		IF fbSQLDatabaseEvt.CreateSP('[dbo].[GetResourcesByNameMilling]', ADR(SQLSPParameterSize1), SIZEOF(SQLSPParameterSize1), pSQLStoredProcedureEvt[29]) THEN	
			IF fbSQLDatabaseEvt.bError THEN
    	
				iState							:=1340;
			ELSE
				
				iState							:= 350;
			END_IF
		END_IF
		
	350:
		SQLSPParameterSize3[0].sParameterName := '@return';
		SQLSPParameterSize3[0].eParameterType := E_SPParameterType.ReturnValue;
		SQLSPParameterSize3[0].eParameterDataType := E_ColumnType.Integer;
		SQLSPParameterSize3[0].nParameterSize := SIZEOF(DINT);
	
		SQLSPParameterSize3[1].sParameterName := '@StatusFilter';
		SQLSPParameterSize3[1].eParameterType := E_SPParameterType.Input;
		SQLSPParameterSize3[1].eParameterDataType := E_ColumnType.NVarChar;
		SQLSPParameterSize3[1].nParameterSize := SIZEOF(STRING(50));
		                  
		SQLSPParameterSize3[2].sParameterName := '@OrderListJson';
		SQLSPParameterSize3[2].eParameterType := E_SPParameterType.Output;
		SQLSPParameterSize3[2].eParameterDataType := E_ColumnType.NVarChar;
		SQLSPParameterSize3[2].nParameterSize := SIZEOF(STRING(DB.MAX_STRING_SIZE));
		
		IF fbSQLDatabaseEvt.CreateSP('[dbo].[MES_GetOrderInfoList]', ADR(SQLSPParameterSize3), SIZEOF(SQLSPParameterSize3), pSQLStoredProcedureEvt[31]) THEN	
			IF fbSQLDatabaseEvt.bError THEN
    	
				iState							:=1350;
			ELSE
				
				iState							:= 360;
			END_IF
		END_IF	
		
	360:
		SQLSPParameterSize3[0].sParameterName := '@return';
		SQLSPParameterSize3[0].eParameterType := E_SPParameterType.ReturnValue;
		SQLSPParameterSize3[0].eParameterDataType := E_ColumnType.Integer;
		SQLSPParameterSize3[0].nParameterSize := SIZEOF(DINT);
	
		SQLSPParameterSize3[1].sParameterName := '@OrderReference';
		SQLSPParameterSize3[1].eParameterType := E_SPParameterType.Input;
		SQLSPParameterSize3[1].eParameterDataType := E_ColumnType.NVarChar;
		SQLSPParameterSize3[1].nParameterSize := SIZEOF(STRING(50));
		                  
		SQLSPParameterSize3[2].sParameterName := '@OrderItemsJson';
		SQLSPParameterSize3[2].eParameterType := E_SPParameterType.Output;
		SQLSPParameterSize3[2].eParameterDataType := E_ColumnType.NVarChar;
		SQLSPParameterSize3[2].nParameterSize := SIZEOF(STRING(DB.MAX_STRING_SIZE));
		
		IF fbSQLDatabaseEvt.CreateSP('[dbo].[MES_GetOrderItems]', ADR(SQLSPParameterSize3), SIZEOF(SQLSPParameterSize3), pSQLStoredProcedureEvt[32]) THEN	
			IF fbSQLDatabaseEvt.bError THEN
    	
				iState							:=1360;
			ELSE
				
				iState							:= 370;
			END_IF
		END_IF	
		
	370:
		SQLSPParameterSize2[0].sParameterName := '@return';
		SQLSPParameterSize2[0].eParameterType := E_SPParameterType.ReturnValue;
		SQLSPParameterSize2[0].eParameterDataType := E_ColumnType.Integer;
		SQLSPParameterSize2[0].nParameterSize := SIZEOF(DINT);
	                      
		SQLSPParameterSize2[1].sParameterName := '@BatchId';
		SQLSPParameterSize2[1].eParameterType := E_SPParameterType.Input;
		SQLSPParameterSize2[1].eParameterDataType := E_ColumnType.NVarChar;
		SQLSPParameterSize2[1].nParameterSize := SIZEOF(STRING(50));
		
		IF fbSQLDatabaseEvt.CreateSP('[dbo].[GetOrderItems]', ADR(SQLSPParameterSize2), SIZEOF(SQLSPParameterSize2), pSQLStoredProcedureEvt[33]) THEN	
			IF fbSQLDatabaseEvt.bError THEN
    	
				iState							:=1370;
			ELSE
				
				iState							:= 380;
			END_IF
		END_IF	
		
	380:
		SQLSPParameterSize3[0].sParameterName := '@return';
		SQLSPParameterSize3[0].eParameterType := E_SPParameterType.ReturnValue;
		SQLSPParameterSize3[0].eParameterDataType := E_ColumnType.Integer;
		SQLSPParameterSize3[0].nParameterSize := SIZEOF(DINT);
	                      
		SQLSPParameterSize3[1].sParameterName := '@InputJson';
		SQLSPParameterSize3[1].eParameterType := E_SPParameterType.Input;
		SQLSPParameterSize3[1].eParameterDataType := E_ColumnType.NVarChar;
		SQLSPParameterSize3[1].nParameterSize := SIZEOF(STRING(DB.MAX_STRING_SIZE));
		
		SQLSPParameterSize3[2].sParameterName := '@OutputJson';
		SQLSPParameterSize3[2].eParameterType := E_SPParameterType.Output;
		SQLSPParameterSize3[2].eParameterDataType := E_ColumnType.NVarChar;
		SQLSPParameterSize3[2].nParameterSize := SIZEOF(STRING(DB.MAX_STRING_SIZE));
	
		IF fbSQLDatabaseEvt.CreateSP('[dbo].[GetBatchList]', ADR(SQLSPParameterSize3), SIZEOF(SQLSPParameterSize3), pSQLStoredProcedureEvt[34]) THEN	
			IF fbSQLDatabaseEvt.bError THEN
    	
				iState							:=1380;
			ELSE
				
				iState							:= 390;
			END_IF
		END_IF
		
	390:
		SQLSPParameterSize3[0].sParameterName := '@return';
		SQLSPParameterSize3[0].eParameterType := E_SPParameterType.ReturnValue;
		SQLSPParameterSize3[0].eParameterDataType := E_ColumnType.Integer;
		SQLSPParameterSize3[0].nParameterSize := SIZEOF(DINT);
	                      
		SQLSPParameterSize3[1].sParameterName := '@InputJson';
		SQLSPParameterSize3[1].eParameterType := E_SPParameterType.Input;
		SQLSPParameterSize3[1].eParameterDataType := E_ColumnType.NVarChar;
		SQLSPParameterSize3[1].nParameterSize := SIZEOF(STRING(DB.MAX_STRING_SIZE));
		
		SQLSPParameterSize3[2].sParameterName := '@OutputJson';
		SQLSPParameterSize3[2].eParameterType := E_SPParameterType.Output;
		SQLSPParameterSize3[2].eParameterDataType := E_ColumnType.NVarChar;
		SQLSPParameterSize3[2].nParameterSize := SIZEOF(STRING(DB.MAX_STRING_SIZE));
	
		IF fbSQLDatabaseEvt.CreateSP('[dbo].[GetBatchList]', ADR(SQLSPParameterSize3), SIZEOF(SQLSPParameterSize3), pSQLStoredProcedureEvt[35]) THEN	
			IF fbSQLDatabaseEvt.bError THEN
    	
				iState							:=1390;
			ELSE
				
				iState							:= 400;
			END_IF
		END_IF
		
	400:
		SQLSPParameterSize1[0].sParameterName := '@return';
		SQLSPParameterSize1[0].eParameterType := E_SPParameterType.ReturnValue;
		SQLSPParameterSize1[0].eParameterDataType := E_ColumnType.Integer;
		SQLSPParameterSize1[0].nParameterSize := SIZEOF(DINT);
		
		IF fbSQLDatabaseEvt.CreateSP('[dbo].[CMD_AbortProduction]', ADR(SQLSPParameterSize1), SIZEOF(SQLSPParameterSize1), pSQLStoredProcedureEvt[36]) THEN	
			IF fbSQLDatabaseEvt.bError THEN
    	
				iState							:=1400;
			ELSE
				
				iState							:= 410;
			END_IF
		END_IF
		
	410:
		SQLSPParameterSize3[0].sParameterName := '@return';
		SQLSPParameterSize3[0].eParameterType := E_SPParameterType.ReturnValue;
		SQLSPParameterSize3[0].eParameterDataType := E_ColumnType.Integer;
		SQLSPParameterSize3[0].nParameterSize := SIZEOF(DINT);
		                  
		SQLSPParameterSize3[1].sParameterName := '@currentPage';
		SQLSPParameterSize3[1].eParameterType := E_SPParameterType.Input;
		SQLSPParameterSize3[1].eParameterDataType := E_ColumnType.Integer;
		SQLSPParameterSize3[1].nParameterSize := SIZEOF(DINT);
		                  
		SQLSPParameterSize3[2].sParameterName := '@recordToFetch';
		SQLSPParameterSize3[2].eParameterType := E_SPParameterType.Input;
		SQLSPParameterSize3[2].eParameterDataType := E_ColumnType.Integer;
		SQLSPParameterSize3[2].nParameterSize := SIZEOF(DINT);
		
		IF fbSQLDatabaseEvt.CreateSP('[dbo].[GetBatchHistory]', ADR(SQLSPParameterSize3), SIZEOF(SQLSPParameterSize3), pSQLStoredProcedureEvt[37]) THEN	
			IF fbSQLDatabaseEvt.bError THEN
    	
				iState							:=1410;
			ELSE
				
				iState							:= 420;
			END_IF
		END_IF

	420:
		SQLSPParameterSize2[0].sParameterName := '@return';
		SQLSPParameterSize2[0].eParameterType := E_SPParameterType.ReturnValue;
		SQLSPParameterSize2[0].eParameterDataType := E_ColumnType.Integer;
		SQLSPParameterSize2[0].nParameterSize := SIZEOF(DINT);

		SQLSPParameterSize2[1].sParameterName := '@BatchId';
		SQLSPParameterSize2[1].eParameterType := E_SPParameterType.Input;
		SQLSPParameterSize2[1].eParameterDataType := E_ColumnType.NVarChar;
		SQLSPParameterSize2[1].nParameterSize := SIZEOF(STRING(50));
		
		IF fbSQLDatabaseEvt.CreateSP('[dbo].[GetBatchHistoryDetail]', ADR(SQLSPParameterSize2), SIZEOF(SQLSPParameterSize2), pSQLStoredProcedureEvt[38]) THEN	
			IF fbSQLDatabaseEvt.bError THEN
    	
				iState							:=1420;
			ELSE
				
				iState							:= 430;
			END_IF
		END_IF
		
	430:
		SQLSPParameterSize2[0].sParameterName := '@return';
		SQLSPParameterSize2[0].eParameterType := E_SPParameterType.ReturnValue;
		SQLSPParameterSize2[0].eParameterDataType := E_ColumnType.Integer;
		SQLSPParameterSize2[0].nParameterSize := SIZEOF(DINT);

		SQLSPParameterSize2[1].sParameterName := '@Id';
		SQLSPParameterSize2[1].eParameterType := E_SPParameterType.Input;
		SQLSPParameterSize2[1].eParameterDataType := E_ColumnType.NVarChar;
		SQLSPParameterSize2[1].nParameterSize := SIZEOF(STRING(50));
		
		IF fbSQLDatabaseEvt.CreateSP('[dbo].[CMD_ForceCompletedBatch]', ADR(SQLSPParameterSize2), SIZEOF(SQLSPParameterSize2), pSQLStoredProcedureEvt[39]) THEN	
			IF fbSQLDatabaseEvt.bError THEN
    	
				iState							:=1430;
			ELSE
				
				iState							:= 440;
			END_IF
		END_IF
		
	440:
		SQLSPParameterSize2[0].sParameterName := '@return';
		SQLSPParameterSize2[0].eParameterType := E_SPParameterType.ReturnValue;
		SQLSPParameterSize2[0].eParameterDataType := E_ColumnType.Integer;
		SQLSPParameterSize2[0].nParameterSize := SIZEOF(DINT);

		SQLSPParameterSize2[1].sParameterName := '@Id';
		SQLSPParameterSize2[1].eParameterType := E_SPParameterType.Input;
		SQLSPParameterSize2[1].eParameterDataType := E_ColumnType.NVarChar;
		SQLSPParameterSize2[1].nParameterSize := SIZEOF(STRING(50));
		
		IF fbSQLDatabaseEvt.CreateSP('[dbo].[CMD_HoldBatch]', ADR(SQLSPParameterSize2), SIZEOF(SQLSPParameterSize2), pSQLStoredProcedureEvt[40]) THEN	
			IF fbSQLDatabaseEvt.bError THEN
    	
				iState							:=1440;
			ELSE
				
				iState							:= 450;
			END_IF
		END_IF
		
	450:
		SQLSPParameterSize3[0].sParameterName := '@return';
		SQLSPParameterSize3[0].eParameterType := E_SPParameterType.ReturnValue;
		SQLSPParameterSize3[0].eParameterDataType := E_ColumnType.Integer;
		SQLSPParameterSize3[0].nParameterSize := SIZEOF(DINT);
                          
		SQLSPParameterSize3[1].sParameterName := '@Id';
		SQLSPParameterSize3[1].eParameterType := E_SPParameterType.Input;
		SQLSPParameterSize3[1].eParameterDataType := E_ColumnType.NVarChar;
		SQLSPParameterSize3[1].nParameterSize := SIZEOF(STRING(50));
		
		SQLSPParameterSize3[2].sParameterName := '@Mode';
		SQLSPParameterSize3[2].eParameterType := E_SPParameterType.Input;
		SQLSPParameterSize3[2].eParameterDataType := E_ColumnType.NVarChar;
		SQLSPParameterSize3[2].nParameterSize := SIZEOF(STRING(50));
		
		IF fbSQLDatabaseEvt.CreateSP('[dbo].[CMD_RecoverBatch]', ADR(SQLSPParameterSize3), SIZEOF(SQLSPParameterSize3), pSQLStoredProcedureEvt[41]) THEN	
			IF fbSQLDatabaseEvt.bError THEN
    	
				iState							:=1450;
			ELSE
				
				iState							:= 460;
			END_IF
		END_IF
		
	460:
		SQLSPParameterSize4[0].sParameterName := '@return';
		SQLSPParameterSize4[0].eParameterType := E_SPParameterType.ReturnValue;
		SQLSPParameterSize4[0].eParameterDataType := E_ColumnType.Integer;
		SQLSPParameterSize4[0].nParameterSize := SIZEOF(DINT);
                          
		SQLSPParameterSize4[1].sParameterName := '@Id';
		SQLSPParameterSize4[1].eParameterType := E_SPParameterType.Input;
		SQLSPParameterSize4[1].eParameterDataType := E_ColumnType.NVarChar;
		SQLSPParameterSize4[1].nParameterSize := SIZEOF(STRING(50));
		                  
		SQLSPParameterSize4[2].sParameterName := '@Mode';
		SQLSPParameterSize4[2].eParameterType := E_SPParameterType.Input;
		SQLSPParameterSize4[2].eParameterDataType := E_ColumnType.NVarChar;
		SQLSPParameterSize4[2].nParameterSize := SIZEOF(STRING(50));
		                  
		SQLSPParameterSize4[3].sParameterName := '@RestartMode';
		SQLSPParameterSize4[3].eParameterType := E_SPParameterType.Input;
		SQLSPParameterSize4[3].eParameterDataType := E_ColumnType.NVarChar;
		SQLSPParameterSize4[3].nParameterSize := SIZEOF(STRING(50));
		
		IF fbSQLDatabaseEvt.CreateSP('[dbo].[CMD_RestartBatch]', ADR(SQLSPParameterSize4), SIZEOF(SQLSPParameterSize4), pSQLStoredProcedureEvt[42]) THEN	
			IF fbSQLDatabaseEvt.bError THEN
    	
				iState							:=1460;
			ELSE
				
				iState							:= 470;
			END_IF
		END_IF
		
	470:
		SQLSPParameterSize3[0].sParameterName := '@return';
		SQLSPParameterSize3[0].eParameterType := E_SPParameterType.ReturnValue;
		SQLSPParameterSize3[0].eParameterDataType := E_ColumnType.Integer;
		SQLSPParameterSize3[0].nParameterSize := SIZEOF(DINT);
                          
		SQLSPParameterSize3[1].sParameterName := '@Id';
		SQLSPParameterSize3[1].eParameterType := E_SPParameterType.Input;
		SQLSPParameterSize3[1].eParameterDataType := E_ColumnType.NVarChar;
		SQLSPParameterSize3[1].nParameterSize := SIZEOF(STRING(50));
		
		SQLSPParameterSize3[2].sParameterName := '@Mode';
		SQLSPParameterSize3[2].eParameterType := E_SPParameterType.Input;
		SQLSPParameterSize3[2].eParameterDataType := E_ColumnType.NVarChar;
		SQLSPParameterSize3[2].nParameterSize := SIZEOF(STRING(50));
		
		IF fbSQLDatabaseEvt.CreateSP('[dbo].[CMD_ResumeBatch]', ADR(SQLSPParameterSize3), SIZEOF(SQLSPParameterSize3), pSQLStoredProcedureEvt[43]) THEN	
			IF fbSQLDatabaseEvt.bError THEN
    	
				iState							:=1470;
			ELSE
				
				iState							:= 480;
			END_IF
		END_IF
		
	480:
		SQLSPParameterSize3[0].sParameterName := '@return';
		SQLSPParameterSize3[0].eParameterType := E_SPParameterType.ReturnValue;
		SQLSPParameterSize3[0].eParameterDataType := E_ColumnType.Integer;
		SQLSPParameterSize3[0].nParameterSize := SIZEOF(DINT);
                          
		SQLSPParameterSize3[1].sParameterName := '@Id';
		SQLSPParameterSize3[1].eParameterType := E_SPParameterType.Input;
		SQLSPParameterSize3[1].eParameterDataType := E_ColumnType.NVarChar;
		SQLSPParameterSize3[1].nParameterSize := SIZEOF(STRING(50));
		
		SQLSPParameterSize3[2].sParameterName := '@Mode';
		SQLSPParameterSize3[2].eParameterType := E_SPParameterType.Input;
		SQLSPParameterSize3[2].eParameterDataType := E_ColumnType.NVarChar;
		SQLSPParameterSize3[2].nParameterSize := SIZEOF(STRING(50));
		
		IF fbSQLDatabaseEvt.CreateSP('[dbo].[CMD_SuspendBatch]', ADR(SQLSPParameterSize3), SIZEOF(SQLSPParameterSize3), pSQLStoredProcedureEvt[44]) THEN	
			IF fbSQLDatabaseEvt.bError THEN
    	
				iState							:=1480;
			ELSE
				
				iState							:= 490;
			END_IF
		END_IF
		
	490:
		SQLSPParameterSize2[0].sParameterName := '@return';
		SQLSPParameterSize2[0].eParameterType := E_SPParameterType.ReturnValue;
		SQLSPParameterSize2[0].eParameterDataType := E_ColumnType.Integer;
		SQLSPParameterSize2[0].nParameterSize := SIZEOF(DINT);

		SQLSPParameterSize2[1].sParameterName := '@Id';
		SQLSPParameterSize2[1].eParameterType := E_SPParameterType.Input;
		SQLSPParameterSize2[1].eParameterDataType := E_ColumnType.NVarChar;
		SQLSPParameterSize2[1].nParameterSize := SIZEOF(STRING(50));
		
		IF fbSQLDatabaseEvt.CreateSP('[dbo].[CMD_UnholdBatch]', ADR(SQLSPParameterSize2), SIZEOF(SQLSPParameterSize2), pSQLStoredProcedureEvt[45]) THEN	
			IF fbSQLDatabaseEvt.bError THEN
    	
				iState							:=1490;
			ELSE
				
				iState							:= 500;
			END_IF
		END_IF

	500:
		SQLSPParameterSize3[0].sParameterName := '@return';
		SQLSPParameterSize3[0].eParameterType := E_SPParameterType.ReturnValue;
		SQLSPParameterSize3[0].eParameterDataType := E_ColumnType.Integer;
		SQLSPParameterSize3[0].nParameterSize := SIZEOF(DINT);

		SQLSPParameterSize3[1].sParameterName := '@Name';
		SQLSPParameterSize3[1].eParameterType := E_SPParameterType.Input;
		SQLSPParameterSize3[1].eParameterDataType := E_ColumnType.NVarChar;
		SQLSPParameterSize3[1].nParameterSize := SIZEOF(STRING(50));
		
		SQLSPParameterSize3[2].sParameterName := '@JsonValue';
		SQLSPParameterSize3[2].eParameterType := E_SPParameterType.Input;
		SQLSPParameterSize3[2].eParameterDataType := E_ColumnType.NVarChar;
		SQLSPParameterSize3[2].nParameterSize := SIZEOF(STRING(DB.MAX_STRING_SIZE));
		
		IF fbSQLDatabaseEvt.CreateSP('[dbo].[UpdateSettingRepositoryByName]', ADR(SQLSPParameterSize3), SIZEOF(SQLSPParameterSize3), pSQLStoredProcedureEvt[46]) THEN	
			IF fbSQLDatabaseEvt.bError THEN
    	
				iState							:=1500;
			ELSE
				
				iState							:= 510;
			END_IF
		END_IF		
	
	510:
		SQLSPParameterSize1[0].sParameterName := '@return';
		SQLSPParameterSize1[0].eParameterType := E_SPParameterType.ReturnValue;
		SQLSPParameterSize1[0].eParameterDataType := E_ColumnType.Integer;
		SQLSPParameterSize1[0].nParameterSize := SIZEOF(DINT);
		
		IF fbSQLDatabaseEvt.CreateSP('[dbo].[GetSettingRepositoryList]', ADR(SQLSPParameterSize1), SIZEOF(SQLSPParameterSize1), pSQLStoredProcedureEvt[47]) THEN	
			IF fbSQLDatabaseEvt.bError THEN
    	
				iState							:=1510;
			ELSE
				
				iState							:= 520;
			END_IF
		END_IF	
		
	520:
		SQLSPParameterSize2[0].sParameterName := '@return';
		SQLSPParameterSize2[0].eParameterType := E_SPParameterType.ReturnValue;
		SQLSPParameterSize2[0].eParameterDataType := E_ColumnType.Integer;
		SQLSPParameterSize2[0].nParameterSize := SIZEOF(DINT);

		SQLSPParameterSize2[1].sParameterName := '@BatchId';
		SQLSPParameterSize2[1].eParameterType := E_SPParameterType.Input;
		SQLSPParameterSize2[1].eParameterDataType := E_ColumnType.NVarChar;
		SQLSPParameterSize2[1].nParameterSize := SIZEOF(STRING(50));
		
		IF fbSQLDatabaseEvt.CreateSP('[dbo].[GetBatchDetailById]', ADR(SQLSPParameterSize2), SIZEOF(SQLSPParameterSize2), pSQLStoredProcedureEvt[48]) THEN	
			IF fbSQLDatabaseEvt.bError THEN
    	
				iState							:=1520;
			ELSE
				
				iState							:=530;
			END_IF
		END_IF
		
	530:
		SQLSPParameterSize3[0].sParameterName := '@return';
		SQLSPParameterSize3[0].eParameterType := E_SPParameterType.ReturnValue;
		SQLSPParameterSize3[0].eParameterDataType := E_ColumnType.Integer;
		SQLSPParameterSize3[0].nParameterSize := SIZEOF(DINT);

		SQLSPParameterSize3[1].sParameterName := '@BatchId';
		SQLSPParameterSize3[1].eParameterType := E_SPParameterType.Input;
		SQLSPParameterSize3[1].eParameterDataType := E_ColumnType.NVarChar;
		SQLSPParameterSize3[1].nParameterSize := SIZEOF(STRING(50));
		
		SQLSPParameterSize3[2].sParameterName := '@DestinationPosition';
		SQLSPParameterSize3[2].eParameterType := E_SPParameterType.Input;
		SQLSPParameterSize3[2].eParameterDataType := E_ColumnType.Integer;
		SQLSPParameterSize3[2].nParameterSize := SIZEOF(DINT);
		
		IF fbSQLDatabaseEvt.CreateSP('[dbo].[ChangeBatchPositionInProductionQueue]', ADR(SQLSPParameterSize3), SIZEOF(SQLSPParameterSize3), pSQLStoredProcedureEvt[49]) THEN	
			IF fbSQLDatabaseEvt.bError THEN
    	
				iState							:=1530;
			ELSE
				
				iState							:= 540;
			END_IF
		END_IF
		
	540:
		SQLSPParameterSize2[0].sParameterName := '@Drum';
		SQLSPParameterSize2[0].eParameterType := E_SPParameterType.Input;
		SQLSPParameterSize2[0].eParameterDataType := E_ColumnType.NVarChar;
		SQLSPParameterSize2[0].nParameterSize := SIZEOF(STRING(30));	
	                      
		SQLSPParameterSize2[1].sParameterName := '@JsonResult';
		SQLSPParameterSize2[1].eParameterType := E_SPParameterType.Output;
		SQLSPParameterSize2[1].eParameterDataType := E_ColumnType.NVarChar;
		SQLSPParameterSize2[1].nParameterSize := SIZEOF(STRING(DB.MAX_STRING_SIZE));
	
		IF fbSQLDatabaseEvt.CreateSP('[dbo].[GetCuttersOnDrum]', ADR(SQLSPParameterSize2), SIZEOF(SQLSPParameterSize2), pSQLStoredProcedureEvt[50]) THEN	
			IF fbSQLDatabaseEvt.bError THEN
    	
				iState							:=1540;
			ELSE
				
				iState							:= 550;
			END_IF
		END_IF
		
	550:
		SQLSPParameterSize1[0].sParameterName := '@JsonResult';
		SQLSPParameterSize1[0].eParameterType := E_SPParameterType.Output;
		SQLSPParameterSize1[0].eParameterDataType := E_ColumnType.NVarChar;
		SQLSPParameterSize1[0].nParameterSize := SIZEOF(STRING(DB.MAX_STRING_SIZE));
	
		IF fbSQLDatabaseEvt.CreateSP('[dbo].[GetCuttersComboboxFormatted]', ADR(SQLSPParameterSize1), SIZEOF(SQLSPParameterSize1), pSQLStoredProcedureEvt[51]) THEN	
			IF fbSQLDatabaseEvt.bError THEN
    	
				iState							:=1550;
			ELSE
				
				iState							:= 560;
			END_IF
		END_IF
		
	560:
		SQLSPParameterSize2[0].sParameterName := '@Drum';
		SQLSPParameterSize2[0].eParameterType := E_SPParameterType.Input;
		SQLSPParameterSize2[0].eParameterDataType := E_ColumnType.NVarChar;
		SQLSPParameterSize2[0].nParameterSize := SIZEOF(STRING(30));	
	                      
		SQLSPParameterSize2[1].sParameterName := '@JsonValue';
		SQLSPParameterSize2[1].eParameterType := E_SPParameterType.Input;
		SQLSPParameterSize2[1].eParameterDataType := E_ColumnType.NVarChar;
		SQLSPParameterSize2[1].nParameterSize := SIZEOF(STRING(DB.MAX_STRING_SIZE));
	
		IF fbSQLDatabaseEvt.CreateSP('[dbo].[UpdateCuttersOnDrum]', ADR(SQLSPParameterSize2), SIZEOF(SQLSPParameterSize2), pSQLStoredProcedureEvt[52]) THEN	
			IF fbSQLDatabaseEvt.bError THEN
    	
				iState							:=1560;
			ELSE
				
				iState							:= 570;
			END_IF
		END_IF
		
	570:
		SQLSPParameterSize3[0].sParameterName := '@Id';
		SQLSPParameterSize3[0].eParameterType := E_SPParameterType.Input;
		SQLSPParameterSize3[0].eParameterDataType := E_ColumnType.Integer;
		SQLSPParameterSize3[0].nParameterSize := SIZEOF(DINT);
		
		SQLSPParameterSize3[1].sParameterName := '@Drum';
		SQLSPParameterSize3[1].eParameterType := E_SPParameterType.Input;
		SQLSPParameterSize3[1].eParameterDataType := E_ColumnType.NVarChar;
		SQLSPParameterSize3[1].nParameterSize := SIZEOF(STRING(30));
                          
		SQLSPParameterSize3[2].sParameterName := '@BatchId';
		SQLSPParameterSize3[2].eParameterType := E_SPParameterType.Output;
		SQLSPParameterSize3[2].eParameterDataType := E_ColumnType.Integer;
		SQLSPParameterSize3[2].nParameterSize := SIZEOF(DINT);
		
		IF fbSQLDatabaseEvt.CreateSP('[dbo].[CheckCutterAlreadyPresentOnDrums]', ADR(SQLSPParameterSize3), SIZEOF(SQLSPParameterSize3), pSQLStoredProcedureEvt[53]) THEN	
			IF fbSQLDatabaseEvt.bError THEN
    	
				iState							:=1570;
			ELSE
				
				iState							:= 580;
			END_IF
		END_IF

	580:
		SQLSPParameterSize2[0].sParameterName := '@Id';
		SQLSPParameterSize2[0].eParameterType := E_SPParameterType.Input;
		SQLSPParameterSize2[0].eParameterDataType := E_ColumnType.Integer;
		SQLSPParameterSize2[0].nParameterSize := SIZEOF(DINT);	
	                      
		SQLSPParameterSize2[1].sParameterName := '@Data';
		SQLSPParameterSize2[1].eParameterType := E_SPParameterType.Input;
		SQLSPParameterSize2[1].eParameterDataType := E_ColumnType.NVarChar;
		SQLSPParameterSize2[1].nParameterSize := SIZEOF(STRING(DB.MAX_STRING_SIZE));
	
		IF fbSQLDatabaseEvt.CreateSP('[dbo].[UpdateCutterData]', ADR(SQLSPParameterSize2), SIZEOF(SQLSPParameterSize2), pSQLStoredProcedureEvt[54]) THEN	
			IF fbSQLDatabaseEvt.bError THEN
    	
				iState							:=1580;
			ELSE
				
				iState							:= 590;
			END_IF
		END_IF

	590:
		SQLSPParameterSize1[0].sParameterName := '@FamilyName';
		SQLSPParameterSize1[0].eParameterType := E_SPParameterType.Input;
		SQLSPParameterSize1[0].eParameterDataType := E_ColumnType.NVarChar;
		SQLSPParameterSize1[0].nParameterSize := SIZEOF(STRING(30));	
	
		IF fbSQLDatabaseEvt.CreateSP('[dbo].[GetProfilesByFamilyName]', ADR(SQLSPParameterSize1), SIZEOF(SQLSPParameterSize1), pSQLStoredProcedureEvt[55]) THEN	
			IF fbSQLDatabaseEvt.bError THEN
    	
				iState							:=1590;
			ELSE
				
				iState							:= 600;
			END_IF
		END_IF		

	600:
		SQLSPParameterSize1[0].sParameterName := '@JsonResultError';
		SQLSPParameterSize1[0].eParameterType := E_SPParameterType.Output;
		SQLSPParameterSize1[0].eParameterDataType := E_ColumnType.NVarChar;
		SQLSPParameterSize1[0].nParameterSize := SIZEOF(STRING(DB.MAX_STRING_SIZE));	

		IF fbSQLDatabaseEvt.CreateSP('[dbo].[GetProfiles]', ADR(SQLSPParameterSize1), SIZEOF(SQLSPParameterSize1), pSQLStoredProcedureEvt[56]) THEN	
			IF fbSQLDatabaseEvt.bError THEN
    	
				iState							:=1600;
			ELSE
				
				iState							:= 610;
			END_IF
		END_IF	
		
	610:
		IF fbSQLDatabaseEvt.CreateSP('[dbo].[GetFamilyNamesForCombobox]', 0, 0, pSQLStoredProcedureEvt[57]) THEN	
			IF fbSQLDatabaseEvt.bError THEN
    	
				iState							:=1610;
			ELSE
				
				iState							:= 620;
			END_IF
		END_IF			
	
	620:
		SQLSPParameterSize2[0].sParameterName := '@FamilyName';
		SQLSPParameterSize2[0].eParameterType := E_SPParameterType.Input;
		SQLSPParameterSize2[0].eParameterDataType := E_ColumnType.NVarChar;
		SQLSPParameterSize2[0].nParameterSize := SIZEOF(STRING(30));	
	                      
		SQLSPParameterSize2[1].sParameterName := '@JsonResult';
		SQLSPParameterSize2[1].eParameterType := E_SPParameterType.Output;
		SQLSPParameterSize2[1].eParameterDataType := E_ColumnType.NVarChar;
		SQLSPParameterSize2[1].nParameterSize := SIZEOF(STRING(DB.MAX_STRING_SIZE));
	
		IF fbSQLDatabaseEvt.CreateSP('[dbo].[GetCuttersFromFamilyName]', ADR(SQLSPParameterSize2), SIZEOF(SQLSPParameterSize2), pSQLStoredProcedureEvt[58]) THEN	
			IF fbSQLDatabaseEvt.bError THEN
    	
				iState							:=1620;
			ELSE
				
				iState							:= 630;
			END_IF
		END_IF	
		
	630:
		SQLSPParameterSize1[0].sParameterName := '@ProfileId';
		SQLSPParameterSize1[0].eParameterType := E_SPParameterType.Input;
		SQLSPParameterSize1[0].eParameterDataType := E_ColumnType.NVarChar;
		SQLSPParameterSize1[0].nParameterSize := SIZEOF(STRING(50));	
	
		IF fbSQLDatabaseEvt.CreateSP('[dbo].[DeleteProfile]', ADR(SQLSPParameterSize1), SIZEOF(SQLSPParameterSize1), pSQLStoredProcedureEvt[59]) THEN	
			IF fbSQLDatabaseEvt.bError THEN
    	
				iState							:=1630;
			ELSE
				
				iState							:= 640;
			END_IF
		END_IF	
		
	640:
		SQLSPParameterSize1[0].sParameterName := '@ProfileData';
		SQLSPParameterSize1[0].eParameterType := E_SPParameterType.Input;
		SQLSPParameterSize1[0].eParameterDataType := E_ColumnType.NVarChar;
		SQLSPParameterSize1[0].nParameterSize := SIZEOF(STRING(DB.MAX_STRING_SIZE));	
	
		IF fbSQLDatabaseEvt.CreateSP('[dbo].[AddProfile]', ADR(SQLSPParameterSize1), SIZEOF(SQLSPParameterSize1), pSQLStoredProcedureEvt[60]) THEN	
			IF fbSQLDatabaseEvt.bError THEN
    	
				iState							:=1640;
			ELSE
				
				iState							:= 650;
			END_IF
		END_IF	
		
	650:
		SQLSPParameterSize1[0].sParameterName := '@CutterId';
		SQLSPParameterSize1[0].eParameterType := E_SPParameterType.Input;
		SQLSPParameterSize1[0].eParameterDataType := E_ColumnType.NVarChar;
		SQLSPParameterSize1[0].nParameterSize := SIZEOF(STRING(50));	
	
		IF fbSQLDatabaseEvt.CreateSP('[dbo].[DeleteCutter]', ADR(SQLSPParameterSize1), SIZEOF(SQLSPParameterSize1), pSQLStoredProcedureEvt[61]) THEN	
			IF fbSQLDatabaseEvt.bError THEN
    	
				iState							:=1650;
			ELSE
				
				iState							:= 660;
			END_IF
		END_IF
		
	660:
		SQLSPParameterSize1[0].sParameterName := '@CutterData';
		SQLSPParameterSize1[0].eParameterType := E_SPParameterType.Input;
		SQLSPParameterSize1[0].eParameterDataType := E_ColumnType.NVarChar;
		SQLSPParameterSize1[0].nParameterSize := SIZEOF(STRING(DB.MAX_STRING_SIZE));	
	
		IF fbSQLDatabaseEvt.CreateSP('[dbo].[AddCutter]', ADR(SQLSPParameterSize1), SIZEOF(SQLSPParameterSize1), pSQLStoredProcedureEvt[62]) THEN	
			IF fbSQLDatabaseEvt.bError THEN
    	
				iState							:=1660;
			ELSE
				
				iState							:= 670;
			END_IF
		END_IF
		
	670:
		IF fbSQLDatabaseEvt.CreateSP('[dbo].[GetBroachingProfileSettings]', 0, 0, pSQLStoredProcedureEvt[63]) THEN	
			IF fbSQLDatabaseEvt.bError THEN
    	
				iState							:=1670;
			ELSE
				
				iState							:= 680;
			END_IF
		END_IF
		
	680:
		SQLSPParameterSize2[0].sParameterName := '@IdBroachingProfileSettings';
		SQLSPParameterSize2[0].eParameterType := E_SPParameterType.Input;
		SQLSPParameterSize2[0].eParameterDataType := E_ColumnType.Integer;
		SQLSPParameterSize2[0].nParameterSize := SIZEOF(DINT);	
	                      
		SQLSPParameterSize2[1].sParameterName := '@DataBroachingProfile';
		SQLSPParameterSize2[1].eParameterType := E_SPParameterType.Input;
		SQLSPParameterSize2[1].eParameterDataType := E_ColumnType.NVarChar;
		SQLSPParameterSize2[1].nParameterSize := SIZEOF(STRING(DB.MAX_STRING_SIZE));
		
		IF fbSQLDatabaseEvt.CreateSP('[dbo].[UpdateBroachingProfileSettings]', ADR(SQLSPParameterSize2), SIZEOF(SQLSPParameterSize2), pSQLStoredProcedureEvt[64]) THEN	
			IF fbSQLDatabaseEvt.bError THEN
    	
				iState							:=1680;
			ELSE
				
				iState							:= 690;
			END_IF
		END_IF
		
	690:
		SQLSPParameterSize6[0].sParameterName := '@return';
		SQLSPParameterSize6[0].eParameterType := E_SPParameterType.ReturnValue;
		SQLSPParameterSize6[0].eParameterDataType := E_ColumnType.Integer;
		SQLSPParameterSize6[0].nParameterSize := SIZEOF(DINT);
	                      
		SQLSPParameterSize6[1].sParameterName := '@EventId';
		SQLSPParameterSize6[1].eParameterType := E_SPParameterType.Input;
		SQLSPParameterSize6[1].eParameterDataType := E_ColumnType.BigInt;
		SQLSPParameterSize6[1].nParameterSize := SIZEOF(LINT);
		                  
		SQLSPParameterSize6[2].sParameterName := '@EventTimeStamp';
		SQLSPParameterSize6[2].eParameterType := E_SPParameterType.Input;
		SQLSPParameterSize6[2].eParameterDataType := E_ColumnType.DateTime;
		SQLSPParameterSize6[2].nParameterSize := SIZEOF(DT);
		                  
		SQLSPParameterSize6[3].sParameterName := '@EventType';
		SQLSPParameterSize6[3].eParameterType := E_SPParameterType.Input;
		SQLSPParameterSize6[3].eParameterDataType := E_ColumnType.Integer;
		SQLSPParameterSize6[3].nParameterSize := SIZEOF(DINT);
		
		SQLSPParameterSize6[4].sParameterName := '@Mode';
		SQLSPParameterSize6[4].eParameterType := E_SPParameterType.Input;
		SQLSPParameterSize6[4].eParameterDataType := E_ColumnType.Integer;
		SQLSPParameterSize6[4].nParameterSize := SIZEOF(DINT);
		
		SQLSPParameterSize6[5].sParameterName := '@State';
		SQLSPParameterSize6[5].eParameterType := E_SPParameterType.Input;
		SQLSPParameterSize6[5].eParameterDataType := E_ColumnType.Integer;
		SQLSPParameterSize6[5].nParameterSize := SIZEOF(DINT);
	
		IF fbSQLDatabaseEvt.CreateSP('[dbo].[LogModeStateEvent]', ADR(SQLSPParameterSize6), SIZEOF(SQLSPParameterSize6), pSQLStoredProcedureEvt[65]) THEN	
			IF fbSQLDatabaseEvt.bError THEN
    	
				iState							:=1690;
			ELSE
				
				iState							:= 700;
			END_IF
		END_IF
		
	700:                        
		SQLSPParameterSize2[0].sParameterName := '@Name';
		SQLSPParameterSize2[0].eParameterType := E_SPParameterType.Input;
		SQLSPParameterSize2[0].eParameterDataType := E_ColumnType.NVarChar;
		SQLSPParameterSize2[0].nParameterSize := SIZEOF(STRING(50));
		                  
		SQLSPParameterSize2[1].sParameterName := '@Data';
		SQLSPParameterSize2[1].eParameterType := E_SPParameterType.Output;
		SQLSPParameterSize2[1].eParameterDataType := E_ColumnType.NVarChar;
		SQLSPParameterSize2[1].nParameterSize := SIZEOF(STRING(DB.MAX_STRING_SIZE));
		
		IF fbSQLDatabaseEvt.CreateSP('[dbo].[GetSettingRepositoryByName]', ADR(SQLSPParameterSize2), SIZEOF(SQLSPParameterSize2), pSQLStoredProcedureEvt[66]) THEN	
			IF fbSQLDatabaseEvt.bError THEN
    	
				iState							:=1700;
			ELSE
				
				iState							:= 710;
			END_IF
		END_IF	
		
	710:
		SQLSPParameterSize1[0].sParameterName := '@return';
		SQLSPParameterSize1[0].eParameterType := E_SPParameterType.ReturnValue;
		SQLSPParameterSize1[0].eParameterDataType := E_ColumnType.Integer;
		SQLSPParameterSize1[0].nParameterSize := SIZEOF(DINT);
		IF fbSQLDatabaseEvt.CreateSP('[dbo].[_TASK1]', ADR(SQLSPParameterSize1), SIZEOF(SQLSPParameterSize1), pSQLStoredProcedureEvt[67]) THEN	
			IF fbSQLDatabaseEvt.bError THEN
    	
				iState							:=1710;
			ELSE
				
				iState							:= 720;
			END_IF
		END_IF	
		
	720:
		SQLSPParameterSize1[0].sParameterName := '@return';
		SQLSPParameterSize1[0].eParameterType := E_SPParameterType.ReturnValue;
		SQLSPParameterSize1[0].eParameterDataType := E_ColumnType.Integer;
		SQLSPParameterSize1[0].nParameterSize := SIZEOF(DINT);
		IF fbSQLDatabaseEvt.CreateSP('[dbo].[_TASK2]', ADR(SQLSPParameterSize1), SIZEOF(SQLSPParameterSize1), pSQLStoredProcedureEvt[68]) THEN	
			IF fbSQLDatabaseEvt.bError THEN
    	
				iState							:=1720;
			ELSE
				
				iState							:= 730;
			END_IF
		END_IF	
		
	730:
		SQLSPParameterSize1[0].sParameterName := '@return';
		SQLSPParameterSize1[0].eParameterType := E_SPParameterType.ReturnValue;
		SQLSPParameterSize1[0].eParameterDataType := E_ColumnType.Integer;
		SQLSPParameterSize1[0].nParameterSize := SIZEOF(DINT);
		IF fbSQLDatabaseEvt.CreateSP('[dbo].[_TASK3]', ADR(SQLSPParameterSize1), SIZEOF(SQLSPParameterSize1), pSQLStoredProcedureEvt[69]) THEN	
			IF fbSQLDatabaseEvt.bError THEN
    	
				iState							:=1730;
			ELSE
				
				iState							:= 740;
			END_IF
		END_IF	
		
	740:
		SQLSPParameterSize1[0].sParameterName := '@return';
		SQLSPParameterSize1[0].eParameterType := E_SPParameterType.ReturnValue;
		SQLSPParameterSize1[0].eParameterDataType := E_ColumnType.Integer;
		SQLSPParameterSize1[0].nParameterSize := SIZEOF(DINT);
		IF fbSQLDatabaseEvt.CreateSP('[dbo].[_TASK4]', ADR(SQLSPParameterSize1), SIZEOF(SQLSPParameterSize1), pSQLStoredProcedureEvt[70]) THEN	
			IF fbSQLDatabaseEvt.bError THEN
    	
				iState							:=1740;
			ELSE
				
				iState							:= 750;
			END_IF
		END_IF	
		
	750:
		SQLSPParameterSize1[0].sParameterName := '@return';
		SQLSPParameterSize1[0].eParameterType := E_SPParameterType.ReturnValue;
		SQLSPParameterSize1[0].eParameterDataType := E_ColumnType.Integer;
		SQLSPParameterSize1[0].nParameterSize := SIZEOF(DINT);
		IF fbSQLDatabaseEvt.CreateSP('[dbo].[_TASK5]', ADR(SQLSPParameterSize1), SIZEOF(SQLSPParameterSize1), pSQLStoredProcedureEvt[71]) THEN	
			IF fbSQLDatabaseEvt.bError THEN
    	
				iState							:=1750;
			ELSE
				
				iState							:= 980;
			END_IF
		END_IF	
	
	
// Connected output state
	980:
		IF fbSQLDatabaseEvt.bConnected THEN
			 Connected := TRUE;
		END_IF

// Disconnected output state		
	990:
		IF(fbSQLDatabaseEvt.Disconnect()) THEN
			Connected := FALSE;
			IF fbSQLDatabaseEvt.bError THEN
				Error						:= TRUE;
				ErrorID						:= 1003;
			ELSE
				
				iState							:= 999;
			END_IF
		END_IF

// Wait for disconnection		
	999:
		;
END_CASE




IF iState > 1000 THEN
	Error := TRUE;
ELSE
	Error := FALSE;
END_IF

END_PROGRAM

// ---- FBs/Database/PRG_MSSQL_UpdatePartLocationsAndProcessingData.TcPOU
PROGRAM PRG_MSSQL_UpdatePartLocationsAndProcessingData
VAR_INPUT
	Execute					: BOOL;
	Enable					: BOOL;
	stProcessingData		: ARRAY[0..CNC.NUM_STATIONS] OF DUT_stProcessingData;
END_VAR
VAR_OUTPUT
	Error					: BOOL;
	ErrorID					: DINT;
	Done					: BOOL;
	Busy					: BOOL;
	ReturnValue				: BOOL;
	tcMessage 				: I_TcMessage;
END_VAR
VAR
	RTRIG_Execute			: R_TRIG;
	iState					: INT := -1;
	fbJsonDataType 			: FB_JsonReadWriteDataType;
	hr	:	HRESULT;
	i	: UINT;
	ArrayElement	: STRING(DB.MAX_STRING_SIZE);
	tempString : STRING;
END_VAR
VAR_IN_OUT
	fbSQLStoredProcedure	: FB_SQLStoredProcedureEvt;
	fbSQLResult				: FB_SQLResultEvt;
	Parameters		: DUT_UpdatePartLocationsAndProcessingData;
END_VAR

RTRIG_Execute(CLK := Execute AND Enable);
IF(RTRIG_Execute.Q) THEN
	 Done	 := FALSE;
	 Error	 := FALSE;
	 ErrorID := 0;
	         
	 iState	 := 0;
ELSIF NOT Execute AND NOT Busy THEN
	Busy			:= FALSE;
	Done			:= FALSE;
	Error			:= FALSE;
	
	iState := -1;
END_IF
 
CASE iState OF
 
	0:
 		ReturnValue	:= FALSE;
		Busy		:= TRUE;
		
		Parameters.Data :='[';
		tempString := ',';
		
		iState 		:= 10;
	
	10:
		// creazione JSON array
		FOR i := 0 TO CNC.NUM_STATIONS DO
			fbJsonDataType.CopyJsonStringFromSymbol('DUT_stProcessingData', SIZEOF(stProcessingData[i]), ADR(stProcessingData[i]), ArrayElement, SIZEOF(ArrayElement), hrErrorCode => hr);
			IF SUCCEEDED(hr) THEN
				CONCAT2(ADR(Parameters.Data), ADR(ArrayElement), ADR(Parameters.Data), SIZEOF(Parameters.Data));
				IF i <> CNC.NUM_STATIONS THEN
					CONCAT2(ADR(Parameters.Data), ADR(tempString), ADR(Parameters.Data), SIZEOF(Parameters.Data));
				END_IF
			ELSE
				iState := 1010;
				RETURN;
			END_IF
		END_FOR
   		
		tempString := ']';
		CONCAT2(ADR(Parameters.Data), ADR(tempString), ADR(Parameters.Data), SIZEOF(Parameters.Data));
		iState := 20;

	20:
		IF fbSQLStoredProcedure.Execute(pParameterStrc := ADR(Parameters), cbParameterStrc:= SIZEOF(Parameters)) THEN
			IF fbSQLStoredProcedure.bError THEN
				tcMessage := fbSQLStoredProcedure.ipTcResult;
				
				iState 							:= 1020; 
			ELSE
				iState 							:= 30; 
			END_IF    
		END_IF

	30: 
		IF Parameters.return_value = 0 THEN
			ReturnValue := TRUE;
			
			iState 							:= 999; 
		END_IF
	
	999:
		Done			:= TRUE;
		Busy			:= FALSE;
	
END_CASE 
 
IF iState > 1000 THEN
	Error 		:= TRUE;
	ErrorID	 	:= iState; 
	Busy	 	:= FALSE;
	iState := -1;
END_IF

END_PROGRAM

// ---- FBs/Database/PRG_MSSQL_spGetProcessingDataForHMI.TcPOU
PROGRAM PRG_MSSQL_spGetProcessingDataForHMI
VAR_INPUT
	Execute					: BOOL;
	Enable					: BOOL;
END_VAR
VAR_OUTPUT
	Error					: BOOL;
	ErrorID					: DINT;
	Done					: BOOL;
	Busy					: BOOL;
	tcMessage 				: I_TcMessage;
	Q_tElapsedTime			: TIME;
	Buffer					: STRING(DB.MAX_STRING_SIZE);
	ProcessingHMIDataLocation	: ARRAY[0..CNC.NUM_DATA_POSITION] OF DUT_stProcessingHMIData1;
	ProcessingHMIDataViewData	: ARRAY[0..CNC.NUM_DATA_POSITION] OF DUT_stProcessingHMIData2;
END_VAR
VAR
	RTRIG_Execute			: R_TRIG;
	iState					: INT := -1;	
	fbJsonDataType 			: FB_JsonReadWriteDataType;
	TempArr					: ARRAY[0..2] OF STRING(DB.MAX_STRING_SIZE);
	Lenght					: UDINT;
	TempSeparetor			: ARRAY[0..1] OF STRING(15);
	TempEnd					: STRING(1);
	hr						: HRESULT;
	i						: UINT;
	fbTempWrite				: FB_WriteTestFile;
	fbFileRename : FB_FileRename;
	tempString1	: T_MaxString;
	tempString2	: T_MaxString;
	tempString3	: T_MaxString;
END_VAR
VAR_IN_OUT
	fbSQLResult				: FB_SQLResultEvt;
	fbSQLStoredProcedure	: FB_SQLStoredProcedureEvt;
	Parameters		: DUT_ProcessingDataForHMI;
END_VAR

fbTempWrite(sData := Parameters.ProcessingData,
			sNetId := EC.sNetId,
			sPathName := 'C:\GSCNext\UtilityBAT\fileTest.txt');
tempString3 := FC_myDTtoString(TO_STRING(G.SystemTime));
tempString1 := CONCAT('C:\GSCNext\UtilityBAT\fileTest', tempString3);
tempString2 := CONCAT(tempString1, '.txt');		
fbFileRename(
    sNetId   := EC.sNetId,
    sOldName := 'C:\GSCNext\UtilityBAT\fileTest.txt',
    sNewName := tempString2,
    ePath    := PATH_GENERIC,
    tTimeout := DEFAULT_ADS_TIMEOUT
);

RTRIG_Execute(CLK := Execute AND Enable);
IF(RTRIG_Execute.Q) THEN
	 Done							:= FALSE;
	 Error							:= FALSE;
	 ErrorID						:= 0; 
	 MEMSET(ADR(ProcessingHMIDataLocation),0,SIZEOF(ProcessingHMIDataLocation));
	 MEMSET(ADR(ProcessingHMIDataViewData),0,SIZEOF(ProcessingHMIDataViewData));
	 MEMSET(ADR(TempArr), 0, SIZEOF(TempArr));

	 iState							:= 0;
ELSIF NOT Execute AND NOT Busy THEN
	Busy			:= FALSE;
	Done			:= FALSE;
	Error			:= FALSE;
	
	iState := -1;
END_IF
CASE iState OF
	
	 0:
		Busy								:= TRUE;
		iState 								:= 10;
		
	10:
		IF fbSQLStoredProcedure.ExecuteDataReturn(pParameterStrc := ADR(Parameters), cbParameterStrc := SIZEOF(Parameters), pSQLDBResult := ADR(fbSqlResult)) THEN
			IF fbSQLStoredProcedure.bError THEN
				tcMessage := fbSQLStoredProcedure.ipTcResult;
				iState 							:= 1010; 
			ELSE	
				iState 							:= 30; 
			END_IF    
		END_IF
		
	20:
		IF fbSQLResult.Read(0, fbSQLResult.nDataCount, ADR(Buffer), SIZEOF(Buffer), FALSE, TRUE) THEN
			IF fbSQLResult.bError THEN
				iState 							:= 1020;
			ELSE
				
				iState 							:= 30;
			END_IF
		END_IF
		
	30: 
		IF fbSQLResult.Release() THEN
			iState 								:= 90;		
		END_IF
		
	40:	
		//Buffer := '[{"LocationId":0,"PartId":7,"ViewData":{"ProductName":"Ankerslot","BatchName":"PRD0000001","RowIndex":"1","RowRunningNo":"7","RowQty":"10","OrderReference":"PRD0000001","Profile":"D0U12","Status":"Fetched","RunningNoOverRowQty":"7\/10"}},{"LocationId":1,"PartId":6,"ViewData":{"ProductName":"Ankerslot","BatchName":"PRD0000001","RowIndex":"1","RowRunningNo":"6","RowQty":"10","OrderReference":"PRD0000001","Profile":"D0U12","Status":"Processing","RunningNoOverRowQty":"6\/10"}},{"LocationId":2,"PartId":5,"ViewData":{"ProductName":"Ankerslot","BatchName":"PRD0000001","RowIndex":"1","RowRunningNo":"5","RowQty":"10","OrderReference":"PRD0000001","Profile":"D0U12","Status":"Processing","RunningNoOverRowQty":"5\/10"}},{"LocationId":3,"PartId":4,"ViewData":{"ProductName":"Ankerslot","BatchName":"PRD0000001","RowIndex":"1","RowRunningNo":"4","RowQty":"10","OrderReference":"PRD0000001","Profile":"D0U12","Status":"Processing","RunningNoOverRowQty":"4\/10"}},{"LocationId":4,"PartId":0},{"LocationId":4,"PartId":0},{"LocationId":5,"PartId":0}]';

		//Lenght := LEN2(ADR(Buffer));
		Lenght := LEN2(ADR(Parameters.ProcessingData));
		IF Lenght <= 0 THEN 
			iState 								:= 1040;	
			RETURN;
		END_IF
		
		// Rimuove il primo carattere '['
		DELETE2(ADR(Parameters.ProcessingData),ADR(TempArr[0]), DB.MAX_STRING_SIZE, 1, 1);
		
		// Rimuove l'ultimo carattere ']'
		DELETE2(ADR(TempArr[0]),ADR(TempArr[0]), DB.MAX_STRING_SIZE, 1, Lenght - 1);
		
		TempEnd := '}';	
		TempSeparetor[0] := '},';	
		TempSeparetor[1] := '"ViewData":';		
		FOR i := 0 TO CNC.NUM_DATA_POSITION DO
			// Estrai singolo oggetto JSON: "LocationId":0,"PartId":0}
			FindAndSplit(ADR(TempSeparetor[0]),ADR(TempArr[0]),ADR(TempArr[0]),DB.MAX_STRING_SIZE,ADR(TempArr[1]), DB.MAX_STRING_SIZE,FALSE);
			
			// Estrai solo la parte ViewData da TempArr[0] solo se presente
			IF FIND2(ADR(TempArr[0]),ADR(TempSeparetor[1])) <> 0 THEN
				FindAndSplit(ADR(TempSeparetor[1]),ADR(TempArr[0]),ADR(TempArr[0]),DB.MAX_STRING_SIZE,ADR(TempArr[2]), DB.MAX_STRING_SIZE,FALSE);
			END_IF
			
			Lenght := LEN2(ADR(TempArr[0]));
			IF Lenght > 0 THEN
				IF i <> CNC.NUM_DATA_POSITION THEN
					
					 // Se termina con virgola la rimuove
					IF TempArr[0][Lenght-1] = 44 THEN
						DELETE2(ADR(TempArr[0]),ADR(TempArr[0]), DB.MAX_STRING_SIZE, 1, Lenght);
					END_IF
					
					// Se non termina con graffa, l'aggiunge
					IF TempArr[0][Lenght-1] <> 125 THEN
						CONCAT2(ADR(TempArr[0]),ADR(TempEnd),ADR(TempArr[0]), DB.MAX_STRING_SIZE);
					END_IF
				END_IF		
				
				fbJsonDataType.SetSymbolFromJson(TempArr[0],'DUT_stProcessingHMIData1', SIZEOF(ProcessingHMIDataLocation[i]), ADR(ProcessingHMIDataLocation[i]), hrErrorCode => hr);
				IF NOT SUCCEEDED(hr) THEN
					iState 								:= 1041;				
					RETURN;
				END_IF
				
				// Solo se esiste ViewData lo converto in DUT
				Lenght := LEN2(ADR(TempArr[2]));
				IF Lenght <> 0 THEN
					IF TempArr[2][Lenght-1] = 125 AND TempArr[2][Lenght-2] = 125 THEN
						DELETE2(ADR(TempArr[2]),ADR(TempArr[2]), DB.MAX_STRING_SIZE, 1, Lenght);
					END_IF
					fbJsonDataType.SetSymbolFromJson(TempArr[2],'DUT_stProcessingHMIData2', SIZEOF(ProcessingHMIDataViewData[i]), ADR(ProcessingHMIDataViewData[i]), hrErrorCode => hr);
					IF NOT SUCCEEDED(hr) THEN
						iState 								:= 120;
						RETURN;
					END_IF
				END_IF
				
				Lenght := LEN2(ADR(TempArr[1]));
				IF Lenght = 0 THEN
					EXIT;
				END_IF
				// Preparazione per il prossimo ciclo
				TempArr[0] := TempArr[1];
				TempArr[1] := '';
				TempArr[2] := '';
			ELSE
				EXIT;
			END_IF
		END_FOR
		
		iState 								:= 999;	

	90:
		fbTempWrite.Execute := TRUE;
		IF fbTempWrite.Done THEN
			fbTempWrite.Execute := FALSE;
			iState 								:= 40;	
		ELSIF fbTempWrite.Error THEN
			fbTempWrite.Execute := FALSE;
			iState 								:= 1043;
		END_IF	
		
	120:
		fbFileRename.bExecute := TRUE;
		IF fbFileRename.bBusy THEN
			iState 								:= 121;	
		END_IF

	121:
		IF NOT  fbFileRename.bBusy THEN
			fbFileRename.bExecute := FALSE;
			iState 								:= 1042;
		ELSIF fbFileRename.bError THEN
			iState 								:= 1044;
		END_IF
		
		
	999:
		Done			:= TRUE;
		Busy			:= FALSE;
		
END_CASE 
 
IF iState > 1000 THEN
	Error 		:= TRUE;
	ErrorID	 	:= iState; 
	Busy	 	:= FALSE;
	iState := -1;
END_IF

END_PROGRAM

// ---- FBs/FB_WriteTestFile.TcPOU
FUNCTION_BLOCK FB_WriteTestFile 
VAR_INPUT
	Execute 	: BOOL;
	sData		: STRING(DB.MAX_STRING_SIZE);
	sNetId		: STRING;
	sPathName	: STRING;
END_VAR
VAR_OUTPUT
	Busy : BOOL;
	Done : BOOL;
	Error : BOOL;
	ErrorID : DINT;
	ErrorSubID : UDINT;
	Q_tElapsedTime	: TIME;
END_VAR
VAR
	iState : DINT := -1;
	fbFileOpen: FB_FileOpen;
	fbFileClose: FB_FileClose;
	fbFileWrite: FB_FileWrite;
	hSrcFile : UINT;
	RTRIG_Execute : R_TRIG;
	TON_TimeElapsed : TON;
	TON_Timeout		: TON;
END_VAR

TON_Timeout(IN := Busy, PT := T#20S);
IF TON_Timeout.Q THEN
	
	iState := 1999;
END_IF

RTRIG_Execute(CLK := Execute);
TON_TimeElapsed(PT:= T#5S);
IF(RTRIG_Execute.Q) THEN
	ErrorID := 0;
	ErrorSubID := 0;
	
	iState := 0;
ELSIF NOT Execute AND NOT Busy THEN
	Busy			:= FALSE;
	Done			:= FALSE;
	Error			:= FALSE;
	
	iState := -1;
END_IF

CASE iState OF
	-1:
		;
	0:
		TON_TimeElapsed.IN := TRUE;
		fbFileOpen.bExecute := TRUE;
		Busy := TRUE;
		iState := 10;
			
	10:
        fbFileOpen.bExecute := FALSE; 
        IF NOT fbFileOpen.bBusy THEN 
        	IF fbFileOpen.bError THEN 
            	ErrorSubID := fbFileOpen.nErrId; 
                iState := 1010;
               ELSE 
                    hSrcFile := fbFileOpen.hFile;
					fbFileWrite.bExecute := TRUE; 
                 	iState := 20;
               END_IF 
          END_IF
		  
	20:
          fbFileWrite.bExecute := FALSE; 
          IF NOT fbFileWrite.bBusy THEN 
               IF fbFileWrite.bError THEN 
                    ErrorSubID := fbFileWrite.nErrId; 
                    iState := 1020;
               ELSE 
				   fbFileClose.bExecute := TRUE;
				   
                   iState := 30;
               END_IF 
          END_IF

	30:
		 fbFileClose.bExecute := FALSE;
		 IF NOT fbFileClose.bBusy THEN 
         	IF fbFileClose.bError THEN 
            	ErrorSubID := TO_DINT(fbFileClose.nErrId);  
            END_IF 
           
			Q_tElapsedTime 		:= TON_TimeElapsed.ET;
			
			TON_TimeElapsed.IN 	:= FALSE;
			
			iState 				:= 999;
          END_IF 

	999:
			Busy	 			:= FALSE;
			Done				:= TRUE;
		
END_CASE

IF(iState > 999 OR TON_TimeElapsed.Q) THEN
	Error 	:= TRUE;
	ErrorID := iState;
	Busy 	:= FALSE;
ELSE
	Error := FALSE;
END_IF

A_Call();

ACTION A_Call:
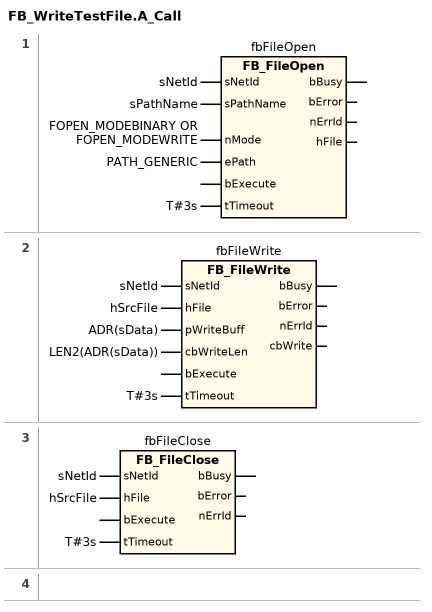
// NETWORK 1
fbFileOpen(
    sNetId := sNetId,
    sPathName := sPathName,
    nMode := FOPEN_MODEBINARY OR FOPEN_MODEWRITE,
    ePath := PATH_GENERIC,
    tTimeout := T#3s); // FB_FileOpen

// NETWORK 2
fbFileWrite(
    sNetId := sNetId,
    hFile := hSrcFile,
    pWriteBuff := ADR(sData),
    cbWriteLen := LEN2(ADR(sData)),
    tTimeout := T#3s); // FB_FileWrite

// NETWORK 3
fbFileClose(sNetId := sNetId, hFile := hSrcFile, tTimeout := T#3s); // FB_FileClose

// NETWORK 4
END_ACTION

END_FUNCTION_BLOCK

// ---- FCs/FC_myDTtoString.TcPOU
FUNCTION FC_myDTtoString : STRING
VAR_INPUT
	in		: STRING;

END_VAR
VAR
	tempString : ARRAY[0..2] OF STRING;
	pos : INT;
END_VAR

tempString[0] := DELETE(in, 3, 1);
pos := FIND(tempString[0], '-');
tempString[1] := tempString[0];
WHILE pos > 0 DO
	tempString[1] := REPLACE(tempString[1], '_', 1, pos);
	pos := FIND(tempString[1], '-');
END_WHILE

pos := FIND(tempString[1], ':');
tempString[2] := tempString[1];
WHILE pos > 0 DO
	tempString[2] := REPLACE(tempString[2], '_', 1, pos);
	pos := FIND(tempString[2], ':');
END_WHILE

FC_myDTtoString := tempString[2];

END_FUNCTION

// ---- FBs/DataRequest/FC_DataFind.TcPOU
FUNCTION FC_DataFind : BOOL
VAR_INPUT
	WIDP : DINT;
	PmcData : POINTER TO DUT_St0Data;
	stPLCData : POINTER TO DUT_stPLCData;
	DataBuffer : POINTER TO DataBuffer;
END_VAR
VAR
	i : UINT;
END_VAR

FC_DataFind := FALSE;
IF WIDP > 0 THEN
	FOR i := 1 TO G.DATABUFFER_SIZE DO
		IF WIDP = DataBuffer[i].WIDP THEN
			PmcData^ := DataBuffer[i].PmcData;
			stPLCData^ := DataBuffer[i].stPLCData;
			FC_DataFind := TRUE;
			RETURN;
		END_IF
	END_FOR	
END_IF

END_FUNCTION

// ---- FBs/DataRequest/FC_UnloadManager.TcPOU
FUNCTION FC_UnloadManager
VAR_IN_OUT
	UnloadingStation : BOOL;
	FLAGP : stByteAsBit;
END_VAR

UnloadingStation := TRUE;
IF FC_ProductStatus(FLAGP) <> eProductStatus.Scraped THEN
	FLAGP.aByte := 0;
	FLAGP.aBit.b0 := 1;
	FLAGP.aBit.b3 := 1;
END_IF

END_FUNCTION

// ---- FCs/FC_OeeSetUpdateCount.TcPOU
FUNCTION FC_OeeSetUpdateCount
VAR_INPUT
	aByte					: stByteAsBit;
END_VAR

IF FC_ProductStatusNopresence(aByte) = eProductStatus.Completed THEN
	G.OEE_bCountUpGood := TRUE;
END_IF
IF FC_ProductStatusNopresence(aByte) = eProductStatus.Scraped THEN
	G.OEE_bCountUpBad := TRUE;
END_IF

END_FUNCTION

// ---- FCs/FC_ProductStatusNoPresence.TcPOU
FUNCTION FC_ProductStatusNoPresence : eProductStatus
VAR_INPUT
	aByte					: stByteAsBit;
END_VAR

IF aByte.aBit.b1 THEN
	FC_ProductStatusNoPresence := eProductStatus.Scraped;
ELSIF aByte.aBit.b3 THEN
	FC_ProductStatusNoPresence := eProductStatus.Completed;
ELSIF aByte.aBit.b2 THEN
	FC_ProductStatusNoPresence := eProductStatus.Working;	
END_IF

END_FUNCTION

// ---- FCs/FC_UpdatePieceCount.TcPOU
FUNCTION FC_UpdatePieceCount
VAR_INPUT
	aByte			: stByteAsBit;
	In				: POINTER TO UDINT;
END_VAR

IF FC_ProductStatusNopresence(aByte) = eProductStatus.Completed THEN
	In[eHeaderPieces.Ok] := In[eHeaderPieces.Ok] + 1;
END_IF
IF FC_ProductStatusNopresence(aByte) = eProductStatus.Scraped THEN
	In[eHeaderPieces.Ko] := In[eHeaderPieces.Ko] + 1;
END_IF

END_FUNCTION

// ---- FCs/FC_BOOLARR_TO_BYTE.TcPOU
FUNCTION FC_BOOLARR_TO_BYTE
VAR_INPUT
	pMyByte : POINTER TO BYTE; // Destination  
	pMyBool : POINTER TO BOOL; // Source   
	nSize	: UINT;               
END_VAR
VAR
    i : UINT;                       
	myByte :  BYTE; 
END_VAR

FOR i:= 0 TO nSize-1 BY 8 DO
	myByte := FC_BOOLBYTE_TO_BYTE(ADR(pMyBool[i]));
	MEMCPY(ADR(pMyByte[i/8]), ADR(myByte), SIZEOF(BYTE));
END_FOR

END_FUNCTION

// ---- FCs/FC_BOOLBYTE_TO_BYTE.TcPOU
FUNCTION FC_BOOLBYTE_TO_BYTE : BYTE
VAR_INPUT
	myBool : POINTER TO BOOL;
END_VAR
VAR
    i : USINT;
END_VAR

FC_BOOLBYTE_TO_BYTE := 0;
FOR i := 0 TO 7 DO
	IF myBool[i] THEN
    	FC_BOOLBYTE_TO_BYTE := FC_BOOLBYTE_TO_BYTE OR (SHL(1,i)) ;
	END_IF
END_FOR

END_FUNCTION

// ---- FBs/FB_TriggerSequencer.TcPOU
FUNCTION_BLOCK FB_TriggerSequencer
VAR_INPUT
    In : ARRAY[0..5] OF BOOL;
    Reset : BOOL;
	Delay : TIME;
END_VAR
VAR_OUTPUT
    Out : BOOL;
END_VAR
VAR
	RTRIG_In : ARRAY[0..5] OF R_TRIG;
	RTRIG_Reset : R_TRIG;
	i : USINT;
	CountPendingTriggers : INT := 0;
	TON_OutDelay	: TON;
END_VAR

TON_OutDelay(PT := Delay);
// Controllo fronti di salita e incremento contatore
FOR i := 0 TO 5 DO
	RTRIG_In[i](CLK := In[i]);
	IF RTRIG_In[i].Q THEN
		CountPendingTriggers := CountPendingTriggers + 1;
	END_IF
END_FOR

// Logica di generazione del trigger
RTRIG_Reset(CLK := Reset);
IF NOT Out AND (CountPendingTriggers > 0) AND NOT Reset THEN
    TON_OutDelay.IN := TRUE;
	IF TON_OutDelay.Q THEN
		TON_OutDelay.IN := FALSE;
		Out := TRUE;
	END_IF
ELSE
    IF RTRIG_Reset.Q AND Out THEN
        CountPendingTriggers := MAX(CountPendingTriggers - 1,0);
        Out := FALSE;
    END_IF
END_IF

END_FUNCTION_BLOCK

// ---- FBs/Database/FB/FB_MSSQL_spGetResourcesByType.TcPOU
FUNCTION_BLOCK FB_MSSQL_spGetResourcesByType
VAR_INPUT
	Execute					: BOOL;
	Enable					: BOOL;
	Reset					: BOOL;
	sType					: STRING(50);
END_VAR
VAR_OUTPUT
	Error					: BOOL;
	ErrorID					: DINT;
	Done					: BOOL;
	Busy					: BOOL;
	tcMessage 				: I_TcMessage;
	Q_tElapsedTime			: TIME;
	Result					: STRING(DB.MAX_STRING_SIZE);
END_VAR
VAR
	RTRIG_Execute			: R_TRIG;
	RTRIG_Reset				: R_TRIG;
	iState					: INT := -1;
	TON_Read				: TON;
	Parameters				: DUT_ResourcesByType;
END_VAR
VAR_IN_OUT
	fbSQLResult				: FB_SQLResultEvt;
	fbSQLStoredProcedure	: FB_SQLStoredProcedureEvt;
END_VAR

RTRIG_Reset(CLK := Reset);
IF RTRIG_Reset.Q AND Execute AND Error AND NOT Busy THEN
	Execute := FALSE;
END_IF

Parameters.ReaourceType :=  sType;
RTRIG_Execute(CLK := Execute AND Enable);
IF(RTRIG_Execute.Q) THEN
	 Done							:= FALSE;
	 Error							:= FALSE;
	 ErrorID						:= 0;
	 
	 iState							:= 0;
ELSIF NOT Execute AND NOT Busy THEN
	Busy			:= FALSE;
	Done			:= FALSE;
	Error			:= FALSE;
	
	iState := -1;
END_IF
 
 // Elapsed Time
 TON_Read(PT:= T#5S);
 
 CASE iState OF
 
	 0:
	 		TON_Read.IN 						:= FALSE;
			Busy								:= TRUE;
			iState 								:= 10;
		
	10:
		IF fbSQLStoredProcedure.ExecuteDataReturn(pParameterStrc := ADR(Parameters), cbParameterStrc:= SIZEOF(Parameters), pSQLDBResult := ADR(fbSqlResult)) THEN
			TON_Read.IN := TRUE;
			IF fbSQLStoredProcedure.bError THEN
				tcMessage := fbSQLStoredProcedure.ipTcResult;
				
				iState 							:= 1010;
			ELSE
				iState 							:= 20;
			END_IF    
		END_IF
		
	20:
		IF fbSQLResult.Read(0, fbSQLResult.nDataCount, ADR(Result), SIZEOF(Result), FALSE, TRUE) THEN
			IF fbSQLResult.bError THEN
				iState 							:= 1020;
			ELSE
			
				iState 							:= 30;
			END_IF
		END_IF
		
	30: 
		IF fbSQLResult.Release() THEN
			iState 								:= 999;	
		END_IF
		
	999:
		TON_Read.IN 	:= FALSE;
		Done			:= TRUE;
		Busy			:= FALSE;
		
 END_CASE 
 
IF iState > 1000 THEN
	Error 		:= TRUE;
	ErrorID	 	:= iState;
	Busy	 	:= FALSE;
	TON_Read.IN := FALSE;
	iState := -1;
END_IF

END_FUNCTION_BLOCK

// ---- FBs/Database/FB/FB_MSSQL_spGetResourcesByName.TcPOU
FUNCTION_BLOCK FB_MSSQL_spGetResourcesByName
VAR_INPUT
	Execute					: BOOL;
	Enable					: BOOL;
	Reset					: BOOL;
	sName					: STRING(50);
END_VAR
VAR_OUTPUT
	Error					: BOOL;
	ErrorID					: DINT;
	Done					: BOOL;
	Busy					: BOOL;
	tcMessage 				: I_TcMessage;
	Q_tElapsedTime			: TIME;
	Result					: STRING(DB.MAX_STRING_SIZE);
END_VAR
VAR
	RTRIG_Execute			: R_TRIG;
	RTRIG_Reset				: R_TRIG;
	iState					: INT := -1;
	TON_Read				: TON;
	Parameters				: DUT_GetResourcesByName;
END_VAR
VAR_IN_OUT
	fbSQLResult				: FB_SQLResultEvt;
	fbSQLStoredProcedure	: FB_SQLStoredProcedureEvt;
END_VAR

RTRIG_Reset(CLK := Reset);
IF RTRIG_Reset.Q AND Execute AND Error AND NOT Busy THEN
	Execute := FALSE;
END_IF

Parameters.ResourceName :=  sName;
RTRIG_Execute(CLK := Execute AND Enable);
IF(RTRIG_Execute.Q) THEN
	 Done							:= FALSE;
	 Error							:= FALSE;
	 ErrorID						:= 0;
	 TON_Read.IN 						:= FALSE;
	 
	 iState							:= 0;
ELSIF NOT Execute AND NOT Busy THEN
	Busy			:= FALSE;
	Done			:= FALSE;
	Error			:= FALSE;
	
	iState := -1;
END_IF
 
 // Elapsed Time
 TON_Read(PT:= T#5S);
 
 CASE iState OF
 
	 0:
			Busy								:= TRUE;
			TON_Read.IN := TRUE;
			iState 								:= 10;
		
	10:
		IF fbSQLStoredProcedure.ExecuteDataReturn(pParameterStrc := ADR(Parameters), cbParameterStrc:= SIZEOF(Parameters), pSQLDBResult := ADR(fbSqlResult)) THEN
			
			IF fbSQLStoredProcedure.bError THEN
				tcMessage := fbSQLStoredProcedure.ipTcResult;
				
				iState 							:= 1010;
			ELSE
				iState 							:= 20;
			END_IF    
		END_IF
		
	20:
		IF fbSQLResult.Read(0, fbSQLResult.nDataCount, ADR(Result), SIZEOF(Result), FALSE, TRUE) THEN
			IF fbSQLResult.bError THEN
				iState 							:= 1020;
			ELSE
				
				iState 							:= 30;
			END_IF
		END_IF
		
	30: 
		IF fbSQLResult.Release() THEN
			Q_tElapsedTime := TON_Read.ET;
			iState 								:= 999;	
		END_IF
		
	999:
		TON_Read.IN 	:= FALSE;
		Done			:= TRUE;
		Busy			:= FALSE;
		
 END_CASE 
 
IF iState > 1000 THEN
	Error 		:= TRUE;
	ErrorID	 	:= iState;
	Busy	 	:= FALSE;
	TON_Read.IN := FALSE;
	iState := -1;
END_IF

END_FUNCTION_BLOCK

// ---- FBs/Database/FB/FB_MSSQL_spSetResourcesByName.TcPOU
FUNCTION_BLOCK FB_MSSQL_spSetResourcesByName
VAR_INPUT
	Execute					: BOOL;
	Enable					: BOOL;
	Reset					: BOOL;
	sName					: STRING(50);
	sNewData				: STRING(DB.MAX_STRING_SIZE);
END_VAR
VAR_OUTPUT
	Error					: BOOL;
	ErrorID					: DINT;
	Done					: BOOL;
	Busy					: BOOL;
	tcMessage 				: I_TcMessage;
	Q_tElapsedTime			: TIME;
	Result					: STRING(DB.MAX_STRING_SIZE);
END_VAR
VAR
	RTRIG_Execute			: R_TRIG;
	RTRIG_Reset				: R_TRIG;
	iState					: INT := -1;
	TON_Read				: TON;
	Parameters				: DUT_SetResourcesByName;
END_VAR
VAR_IN_OUT
	fbSQLStoredProcedure	: FB_SQLStoredProcedureEvt;
END_VAR

RTRIG_Reset(CLK := Reset);
IF RTRIG_Reset.Q AND Execute AND Error AND NOT Busy THEN
	Execute := FALSE;
END_IF

Parameters.ReaourceName :=  sName;
Parameters.NewData :=  sNewData;
RTRIG_Execute(CLK := Execute AND Enable);
IF(RTRIG_Execute.Q) THEN
	 Done							:= FALSE;
	 Error							:= FALSE;
	 ErrorID						:= 0;
	 
	 iState							:= 0;
ELSIF NOT Execute AND NOT Busy THEN
	Busy			:= FALSE;
	Done			:= FALSE;
	Error			:= FALSE;
	
	iState := -1;
END_IF
 
 // Elapsed Time
 TON_Read(PT:= T#5S);
 
 CASE iState OF
 
	 0:
	 		TON_Read.IN 						:= FALSE;
			Busy								:= TRUE;
			iState 								:= 10;
		
	10:
		IF fbSQLStoredProcedure.Execute(pParameterStrc := ADR(Parameters), cbParameterStrc:= SIZEOF(Parameters)) THEN
			TON_Read.IN := TRUE;
			IF fbSQLStoredProcedure.bError THEN
				tcMessage := fbSQLStoredProcedure.ipTcResult;
				
				iState 							:= 1010;
			ELSE
				iState 							:= 999;
			END_IF    
		END_IF
		
	999:
		TON_Read.IN 	:= FALSE;
		Done			:= TRUE;
		Busy			:= FALSE;
		
 END_CASE 
 
IF iState > 1000 THEN
	Error 		:= TRUE;
	ErrorID	 	:= iState;
	Busy	 	:= FALSE;
	TON_Read.IN := FALSE;
	iState := -1;
END_IF

END_FUNCTION_BLOCK

// ---- FBs/Database/FB/FB_MSSQL_spGetResourcesListByType.TcPOU
FUNCTION_BLOCK FB_MSSQL_spGetResourcesListByType
VAR_INPUT
	Execute					: BOOL;
	Enable					: BOOL;
	Reset					: BOOL;
	sType					: STRING(50);
END_VAR
VAR_OUTPUT
	Error					: BOOL;
	ErrorID					: DINT;
	Done					: BOOL;
	Busy					: BOOL;
	tcMessage 				: I_TcMessage;
	Q_tElapsedTime			: TIME;
	Result					: STRING(DB.MAX_STRING_SIZE);
END_VAR
VAR
	RTRIG_Execute			: R_TRIG;
	RTRIG_Reset				: R_TRIG;
	iState					: INT := -1;
	TON_Read				: TON;
	Parameters				: DUT_ResourcesByType;
END_VAR
VAR_IN_OUT
	fbSQLResult				: FB_SQLResultEvt;
	fbSQLStoredProcedure	: FB_SQLStoredProcedureEvt;
END_VAR

RTRIG_Reset(CLK := Reset);
IF RTRIG_Reset.Q AND Execute AND Error AND NOT Busy THEN
	Execute := FALSE;
END_IF

Parameters.ReaourceType :=  sType;
RTRIG_Execute(CLK := Execute AND Enable);
IF(RTRIG_Execute.Q) THEN
	 Done							:= FALSE;
	 Error							:= FALSE;
	 ErrorID						:= 0;
	 
	 iState							:= 0;
ELSIF NOT Execute AND NOT Busy THEN
	Busy			:= FALSE;
	Done			:= FALSE;
	Error			:= FALSE;
	
	iState := -1;
END_IF
 
 // Elapsed Time
 TON_Read(PT:= T#5S);
 
 CASE iState OF
 
	 0:
	 		TON_Read.IN 						:= FALSE;
			Busy								:= TRUE;
			iState 								:= 10;
		
	10:
		IF fbSQLStoredProcedure.ExecuteDataReturn(pParameterStrc := ADR(Parameters), cbParameterStrc:= SIZEOF(Parameters), pSQLDBResult := ADR(fbSqlResult)) THEN
			TON_Read.IN := TRUE;
			IF fbSQLStoredProcedure.bError THEN
				tcMessage := fbSQLStoredProcedure.ipTcResult;
				
				iState 							:= 1010;
			ELSE
				iState 							:= 20;
			END_IF    
		END_IF
		
	20:
		IF fbSQLResult.Read(0, fbSQLResult.nDataCount, ADR(Result), SIZEOF(Result), FALSE, TRUE) THEN
			IF fbSQLResult.bError THEN
				iState 							:= 1020;
			ELSE
			
				iState 							:= 30;
			END_IF
		END_IF
		
	30: 
		IF fbSQLResult.Release() THEN
			iState 								:= 999;	
		END_IF
		
	999:
		TON_Read.IN 	:= FALSE;
		Done			:= TRUE;
		Busy			:= FALSE;
		
 END_CASE 
 
IF iState > 1000 THEN
	Error 		:= TRUE;
	ErrorID	 	:= iState;
	Busy	 	:= FALSE;
	TON_Read.IN := FALSE;
	iState := -1;
END_IF

END_FUNCTION_BLOCK

// ---- FBs/Database/FB/FB_MSSQL_spGetFormattedTablesFromSequences.TcPOU
FUNCTION_BLOCK FB_MSSQL_spGetFormattedTablesFromSequences
VAR_INPUT
	Execute					: BOOL;
	Enable					: BOOL;
	Reset					: BOOL;
	sName					: STRING(50);
END_VAR
VAR_OUTPUT
	Error					: BOOL;
	ErrorID					: DINT;
	Done					: BOOL;
	Busy					: BOOL;
	tcMessage 				: I_TcMessage;
	Q_tElapsedTime			: TIME;
	Result					: STRING(DB.MAX_STRING_SIZE);
END_VAR
VAR
	RTRIG_Execute			: R_TRIG;
	RTRIG_Reset				: R_TRIG;
	iState					: INT := -1;
	TON_Read				: TON;
	Parameters				: DUT_GetResourcesByName;
END_VAR
VAR_IN_OUT
	fbSQLResult				: FB_SQLResultEvt;
	fbSQLStoredProcedure	: FB_SQLStoredProcedureEvt;
END_VAR

RTRIG_Reset(CLK := Reset);
IF RTRIG_Reset.Q AND Execute AND Error AND NOT Busy THEN
	Execute := FALSE;
END_IF

Parameters.ResourceName :=  sName;
RTRIG_Execute(CLK := Execute AND Enable);
IF(RTRIG_Execute.Q) THEN
	 Done							:= FALSE;
	 Error							:= FALSE;
	 ErrorID						:= 0;
	 
	 iState							:= 0;
ELSIF NOT Execute AND NOT Busy THEN
	Busy			:= FALSE;
	Done			:= FALSE;
	Error			:= FALSE;
	
	iState := -1;
END_IF
 
 // Elapsed Time
 TON_Read(PT:= T#5S);
 
 CASE iState OF
 
	 0:
	 		TON_Read.IN 						:= FALSE;
			Busy								:= TRUE;
			iState 								:= 10;
		
	10:
		IF fbSQLStoredProcedure.ExecuteDataReturn(pParameterStrc := ADR(Parameters), cbParameterStrc:= SIZEOF(Parameters), pSQLDBResult := ADR(fbSqlResult)) THEN
			TON_Read.IN := TRUE;
			IF fbSQLStoredProcedure.bError THEN
				tcMessage := fbSQLStoredProcedure.ipTcResult;
				
				iState 							:= 1010;
			ELSE
				iState 							:= 20;
			END_IF    
		END_IF
		
	20:
		IF fbSQLResult.Read(0, fbSQLResult.nDataCount, ADR(Result), SIZEOF(Result), FALSE, TRUE) THEN
			IF fbSQLResult.bError THEN
				iState 							:= 1020;
			ELSE
			
				iState 							:= 30;
			END_IF
		END_IF
		
	30: 
		IF fbSQLResult.Release() THEN
			iState 								:= 999;	
		END_IF
		
	999:
		TON_Read.IN 	:= FALSE;
		Done			:= TRUE;
		Busy			:= FALSE;
		
 END_CASE 
 
IF iState > 1000 THEN
	Error 		:= TRUE;
	ErrorID	 	:= iState;
	Busy	 	:= FALSE;
	TON_Read.IN := FALSE;
	iState := -1;
END_IF

END_FUNCTION_BLOCK

// ---- FBs/Database/FB/FB_MSSQL_spGetOriginsFromSequence.TcPOU
FUNCTION_BLOCK FB_MSSQL_spGetOriginsFromSequence
VAR_INPUT
	Execute					: BOOL;
	Enable					: BOOL;
	Reset					: BOOL;
	sName					: STRING(50);
END_VAR
VAR_OUTPUT
	Error					: BOOL;
	ErrorID					: DINT;
	Done					: BOOL;
	Busy					: BOOL;
	tcMessage 				: I_TcMessage;
	Q_tElapsedTime			: TIME;
	Result					: STRING(DB.MAX_STRING_SIZE);
END_VAR
VAR
	RTRIG_Execute			: R_TRIG;
	RTRIG_Reset				: R_TRIG;
	iState					: INT := -1;
	TON_Read				: TON;
	Parameters				: DUT_SequenceByName;
END_VAR
VAR_IN_OUT
	fbSQLResult				: FB_SQLResultEvt;
	fbSQLStoredProcedure	: FB_SQLStoredProcedureEvt;
END_VAR

RTRIG_Reset(CLK := Reset);
IF RTRIG_Reset.Q AND Execute AND Error AND NOT Busy THEN
	Execute := FALSE;
END_IF

Parameters.SequenceName :=  sName;
RTRIG_Execute(CLK := Execute AND Enable);
IF(RTRIG_Execute.Q) THEN
	 Done							:= FALSE;
	 Error							:= FALSE;
	 ErrorID						:= 0;
	 
	 iState							:= 0;
ELSIF NOT Execute AND NOT Busy THEN
	Busy			:= FALSE;
	Done			:= FALSE;
	Error			:= FALSE;
	
	iState := -1;
END_IF
 
 // Elapsed Time
 TON_Read(PT:= T#5S);
 
 CASE iState OF
 
	 0:
	 		TON_Read.IN 						:= FALSE;
			Busy								:= TRUE;
			iState 								:= 10;
		
	10:
		IF fbSQLStoredProcedure.ExecuteDataReturn(pParameterStrc := ADR(Parameters), cbParameterStrc:= SIZEOF(Parameters), pSQLDBResult := ADR(fbSqlResult)) THEN
			TON_Read.IN := TRUE;
			IF fbSQLStoredProcedure.bError THEN
				tcMessage := fbSQLStoredProcedure.ipTcResult;
				
				iState 							:= 1010;
			ELSE
				iState 							:= 20;
			END_IF    
		END_IF
		
	20:
		IF fbSQLResult.Read(0, fbSQLResult.nDataCount, ADR(Result), SIZEOF(Result), FALSE, TRUE) THEN
			IF fbSQLResult.bError THEN
				iState 							:= 1020;
			ELSE
			
				iState 							:= 30;
			END_IF
		END_IF
		
	30: 
		IF fbSQLResult.Release() THEN
			iState 								:= 999;	
		END_IF
		
	999:
		TON_Read.IN 	:= FALSE;
		Done			:= TRUE;
		Busy			:= FALSE;
		
 END_CASE 
 
IF iState > 1000 THEN
	Error 		:= TRUE;
	ErrorID	 	:= iState;
	Busy	 	:= FALSE;
	TON_Read.IN := FALSE;
	iState := -1;
END_IF

END_FUNCTION_BLOCK

// ---- FBs/Database/FB/FB_MSSQL_spGetBlankKey.TcPOU
FUNCTION_BLOCK FB_MSSQL_spGetBlankKey
VAR_INPUT
	Execute					: BOOL;
	Enable					: BOOL;
	Reset					: BOOL;
END_VAR
VAR_OUTPUT
	Error					: BOOL;
	ErrorID					: DINT;
	Done					: BOOL;
	Busy					: BOOL;
	tcMessage 				: I_TcMessage;
	Q_tElapsedTime			: TIME;
	Result					: STRING(DB.MAX_STRING_SIZE);
END_VAR
VAR
	RTRIG_Execute			: R_TRIG;
	RTRIG_Reset				: R_TRIG;
	iState					: INT := -1;
	TON_Read				: TON;
	return_value	: DINT;
END_VAR
VAR_IN_OUT
	fbSQLResult				: FB_SQLResultEvt;
	fbSQLStoredProcedure	: FB_SQLStoredProcedureEvt;
END_VAR

RTRIG_Reset(CLK := Reset);
IF RTRIG_Reset.Q AND Execute AND Error AND NOT Busy THEN
	Execute := FALSE;
END_IF

RTRIG_Execute(CLK := Execute AND Enable);
IF(RTRIG_Execute.Q) THEN
	 Done							:= FALSE;
	 Error							:= FALSE;
	 ErrorID						:= 0;
	 
	 iState							:= 0;
ELSIF NOT Execute AND NOT Busy THEN
	Busy			:= FALSE;
	Done			:= FALSE;
	Error			:= FALSE;
	
	iState := -1;
END_IF
 
 // Elapsed Time
 TON_Read(PT:= T#5S);
 
 CASE iState OF
 
	 0:
	 		TON_Read.IN 						:= FALSE;
			Busy								:= TRUE;
			iState 								:= 10;
		
	10:
		IF fbSQLStoredProcedure.ExecuteDataReturn(pParameterStrc := ADR(return_value), cbParameterStrc:= SIZEOF(return_value), pSQLDBResult := ADR(fbSqlResult)) THEN
			TON_Read.IN := TRUE;
			IF fbSQLStoredProcedure.bError THEN
				tcMessage := fbSQLStoredProcedure.ipTcResult;
				
				iState 							:= 1010;
			ELSE
				iState 							:= 20;
			END_IF    
		END_IF
		
	20:
		IF fbSQLResult.Read(0, fbSQLResult.nDataCount, ADR(Result), SIZEOF(Result), FALSE, TRUE) THEN
			IF fbSQLResult.bError THEN
				iState 							:= 1020;
			ELSE
				
				iState 							:= 30;
			END_IF
		END_IF
		
	30: 
		IF fbSQLResult.Release() THEN
			iState 								:= 999;	
		END_IF
		
	999:
		TON_Read.IN 	:= FALSE;
		Done			:= TRUE;
		Busy			:= FALSE;
		
 END_CASE 
 
IF iState > 1000 THEN
	Error 		:= TRUE;
	ErrorID	 	:= iState;
	Busy	 	:= FALSE;
	TON_Read.IN := FALSE;
	iState := -1;
END_IF

END_FUNCTION_BLOCK

// ---- FBs/Database/FB/FB_MSSQL_spGetBlankKeyByName.TcPOU
FUNCTION_BLOCK FB_MSSQL_spGetBlankKeyByName
VAR_INPUT
	Execute					: BOOL;
	Enable					: BOOL;
	Reset					: BOOL;
	sName					: STRING(50);
END_VAR
VAR_OUTPUT
	Error					: BOOL;
	ErrorID					: DINT;
	Done					: BOOL;
	Busy					: BOOL;
	tcMessage 				: I_TcMessage;
	Q_tElapsedTime			: TIME;
	Result					: STRING(DB.MAX_STRING_SIZE);
END_VAR
VAR
	RTRIG_Execute			: R_TRIG;
	RTRIG_Reset				: R_TRIG;
	iState					: INT := -1;
	TON_Read				: TON;
	Parameters				: DUT_GetResourcesByName;
END_VAR
VAR_IN_OUT
	fbSQLResult				: FB_SQLResultEvt;
	fbSQLStoredProcedure	: FB_SQLStoredProcedureEvt;
END_VAR

RTRIG_Reset(CLK := Reset);
IF RTRIG_Reset.Q AND Execute AND Error AND NOT Busy THEN
	Execute := FALSE;
END_IF

Parameters.ResourceName :=  sName;
RTRIG_Execute(CLK := Execute AND Enable);
IF(RTRIG_Execute.Q) THEN
	 Done							:= FALSE;
	 Error							:= FALSE;
	 ErrorID						:= 0;
	 
	 iState							:= 0;
ELSIF NOT Execute AND NOT Busy THEN
	Busy			:= FALSE;
	Done			:= FALSE;
	Error			:= FALSE;
	
	iState := -1;
END_IF
 
 // Elapsed Time
 TON_Read(PT:= T#5S);
 
 CASE iState OF
 
	 0:
	 		TON_Read.IN 						:= FALSE;
			Busy								:= TRUE;
			iState 								:= 10;
		
	10:
		IF fbSQLStoredProcedure.ExecuteDataReturn(pParameterStrc := ADR(Parameters), cbParameterStrc:= SIZEOF(Parameters), pSQLDBResult := ADR(fbSqlResult)) THEN
			TON_Read.IN := TRUE;
			IF fbSQLStoredProcedure.bError THEN
				tcMessage := fbSQLStoredProcedure.ipTcResult;
				
				iState 							:= 1010;
			ELSE
				iState 							:= 20;
			END_IF    
		END_IF
		
	20:
		IF fbSQLResult.Read(0, fbSQLResult.nDataCount, ADR(Result), SIZEOF(Result), FALSE, TRUE) THEN
			IF fbSQLResult.bError THEN
				iState 							:= 1020;
			ELSE
				
				iState 							:= 30;
			END_IF
		END_IF
		
	30: 
		IF fbSQLResult.Release() THEN
			iState 								:= 999;	
		END_IF
		
	999:
		TON_Read.IN 	:= FALSE;
		Done			:= TRUE;
		Busy			:= FALSE;
		
 END_CASE 
 
IF iState > 1000 THEN
	Error 		:= TRUE;
	ErrorID	 	:= iState;
	Busy	 	:= FALSE;
	TON_Read.IN := FALSE;
	iState := -1;
END_IF

END_FUNCTION_BLOCK

// ---- FBs/Database/FB/FB_MSSQL_spGetBatchHistory.TcPOU
FUNCTION_BLOCK FB_MSSQL_spGetBatchHistory
VAR_INPUT
	Execute					: BOOL;
	Enable					: BOOL;
	Reset					: BOOL;
	CurrentPage				: DINT;
	RecordToFetch			: DINT;
END_VAR
VAR_OUTPUT
	Error					: BOOL;
	ErrorID					: DINT;
	Done					: BOOL;
	Busy					: BOOL;
	tcMessage 				: I_TcMessage;
	Q_tElapsedTime			: TIME;
	Result					: STRING(DB.MAX_STRING_SIZE);
END_VAR
VAR
	RTRIG_Execute			: R_TRIG;
	RTRIG_Reset				: R_TRIG;
	iState					: INT := -1;
	TON_Read				: TON;
	Parameters		: DUT_GetBatchHistory;
END_VAR
VAR_IN_OUT
	fbSQLResult				: FB_SQLResultEvt;
	fbSQLStoredProcedure	: FB_SQLStoredProcedureEvt;
END_VAR

RTRIG_Reset(CLK := Reset);
IF RTRIG_Reset.Q AND Execute AND Error AND NOT Busy THEN
	Execute := FALSE;
END_IF

Parameters.CurrentPage := CurrentPage;
Parameters.RecordToFetch := RecordToFetch;

RTRIG_Execute(CLK := Execute AND Enable);
IF(RTRIG_Execute.Q) THEN
	 Done							:= FALSE;
	 Error							:= FALSE;
	 ErrorID						:= 0;
	 
	 iState							:= 0;
ELSIF NOT Execute AND NOT Busy THEN
	Busy			:= FALSE;
	Done			:= FALSE;
	Error			:= FALSE;
	
	iState := -1;
END_IF
 
 // Elapsed Time
 TON_Read(PT:= T#5S);
 
 CASE iState OF
 
	 0:
	 		TON_Read.IN 						:= FALSE;
			Busy								:= TRUE;
			iState 								:= 10;
		
	10:
		IF fbSQLStoredProcedure.ExecuteDataReturn(pParameterStrc := ADR(Parameters), cbParameterStrc:= SIZEOF(Parameters), pSQLDBResult := ADR(fbSqlResult)) THEN
			TON_Read.IN := TRUE;
			IF fbSQLStoredProcedure.bError THEN
				tcMessage := fbSQLStoredProcedure.ipTcResult;
				
				iState 							:= 1010;
			ELSE
				iState 							:= 20;
			END_IF    
		END_IF
		
	20:
		IF fbSQLResult.Read(0, fbSQLResult.nDataCount, ADR(Result), SIZEOF(Result), FALSE, TRUE) THEN
			IF fbSQLResult.bError THEN
				iState 							:= 1020;
			ELSE
				
				iState 							:= 30;
			END_IF
		END_IF
		
	30: 
		IF fbSQLResult.Release() THEN
			iState 								:= 999;	
		END_IF
		
	999:
		TON_Read.IN 	:= FALSE;
		Done			:= TRUE;
		Busy			:= FALSE;
		
 END_CASE 
 
IF iState > 1000 THEN
	Error 		:= TRUE;
	ErrorID	 	:= iState;
	Busy	 	:= FALSE;
	TON_Read.IN := FALSE;
	iState := -1;
END_IF

END_FUNCTION_BLOCK

// ---- FBs/Database/FB/FB_MSSQL_spGetBatchHistoryByStatus.TcPOU
FUNCTION_BLOCK FB_MSSQL_spGetBatchHistoryByStatus
VAR_INPUT
	Execute					: BOOL;
	Reset					: BOOL;
	sStatus					: STRING(50);
	Enable					: BOOL;
END_VAR
VAR_OUTPUT
	Error					: BOOL;
	ErrorID					: DINT;
	Done					: BOOL;
	Busy					: BOOL;
	tcMessage 				: I_TcMessage;
	Q_tElapsedTime			: TIME;
	Result					: STRING(DB.MAX_STRING_SIZE);
END_VAR
VAR
	RTRIG_Execute			: R_TRIG;
	RTRIG_Reset				: R_TRIG;
	iState					: INT := -1;
	TON_Read				: TON;
END_VAR
VAR_IN_OUT
	fbSQLResult				: FB_SQLResultEvt;
	fbSQLStoredProcedure	: FB_SQLStoredProcedureEvt;
END_VAR

RTRIG_Reset(CLK := Reset);
IF RTRIG_Reset.Q AND Execute AND Error AND NOT Busy THEN
	Execute := FALSE;
END_IF

RTRIG_Execute(CLK := Execute AND Enable);
IF(RTRIG_Execute.Q) THEN
	 Done							:= FALSE;
	 Error							:= FALSE;
	 ErrorID						:= 0;
	 
	 iState							:= 0;
ELSIF NOT Execute AND NOT Busy THEN
	Busy			:= FALSE;
	Done			:= FALSE;
	Error			:= FALSE;
	
	iState := -1;
END_IF
 
 // Elapsed Time
 TON_Read(PT:= T#5S);
 
 CASE iState OF
 
	 0:
	 		TON_Read.IN 						:= FALSE;
			Busy								:= TRUE;
			iState 								:= 10;
		
	10:
		IF fbSQLStoredProcedure.ExecuteDataReturn(pParameterStrc := ADR(sStatus), cbParameterStrc:= SIZEOF(sStatus), pSQLDBResult := ADR(fbSqlResult)) THEN
			TON_Read.IN := TRUE;
			IF fbSQLStoredProcedure.bError THEN
				tcMessage := fbSQLStoredProcedure.ipTcResult;
				
				iState 							:= 1010;
			ELSE
				iState 							:= 20;
			END_IF    
		END_IF
		
	20:
		IF fbSQLResult.Read(0, fbSQLResult.nDataCount, ADR(Result), SIZEOF(Result), FALSE, TRUE) THEN
			IF fbSQLResult.bError THEN
				iState 							:= 1020;
			ELSE
				
				iState 							:= 30;
			END_IF
		END_IF
		
	30: 
		IF fbSQLResult.Release() THEN
			iState 								:= 999;	
		END_IF
		
	999:
		TON_Read.IN 	:= FALSE;
		Done			:= TRUE;
		Busy			:= FALSE;
		
 END_CASE 
 
IF iState > 1000 THEN
	Error 		:= TRUE;
	ErrorID	 	:= iState;
	Busy	 	:= FALSE;
	TON_Read.IN := FALSE;
	iState := -1;
END_IF

END_FUNCTION_BLOCK

// ---- FBs/Database/FB/FB_MSSQL_spGetPartHistory.TcPOU
FUNCTION_BLOCK FB_MSSQL_spGetPartHistory
VAR_INPUT
	Execute					: BOOL;
	Enable					: BOOL;
	Reset					: BOOL;
END_VAR
VAR_OUTPUT
	Error					: BOOL;
	ErrorID					: DINT;
	Done					: BOOL;
	Busy					: BOOL;
	tcMessage 				: I_TcMessage;
	Q_tElapsedTime			: TIME;
	Result					: STRING(DB.MAX_STRING_SIZE);
END_VAR
VAR
	RTRIG_Execute			: R_TRIG;
	RTRIG_Reset				: R_TRIG;
	iState					: INT := -1;
	TON_Read				: TON;
	return_value	: DINT;
END_VAR
VAR_IN_OUT
	fbSQLResult				: FB_SQLResultEvt;
	fbSQLStoredProcedure	: FB_SQLStoredProcedureEvt;
END_VAR

RTRIG_Reset(CLK := Reset);
IF RTRIG_Reset.Q AND Execute AND Error AND NOT Busy THEN
	Execute := FALSE;
END_IF

RTRIG_Execute(CLK := Execute AND Enable);
IF(RTRIG_Execute.Q) THEN
	 Done							:= FALSE;
	 Error							:= FALSE;
	 ErrorID						:= 0;
	 
	 iState							:= 0;
ELSIF NOT Execute AND NOT Busy THEN
	Busy			:= FALSE;
	Done			:= FALSE;
	Error			:= FALSE;
	
	iState := -1;
END_IF
 
 // Elapsed Time
 TON_Read(PT:= T#5S);
 
 CASE iState OF
 
	 0:
	 		TON_Read.IN 						:= FALSE;
			Busy								:= TRUE;
			iState 								:= 10;
		
	10:
		IF fbSQLStoredProcedure.ExecuteDataReturn(pParameterStrc := 0, cbParameterStrc:= 0, pSQLDBResult := ADR(fbSqlResult)) THEN
			TON_Read.IN := TRUE;
			IF fbSQLStoredProcedure.bError THEN
				tcMessage := fbSQLStoredProcedure.ipTcResult;
				
				iState 							:= 1010;
			ELSE
				iState 							:= 20;
			END_IF    
		END_IF
		
	20:
		IF fbSQLResult.Read(0, fbSQLResult.nDataCount, ADR(Result), SIZEOF(Result), FALSE, TRUE) THEN
			IF fbSQLResult.bError THEN
				iState 							:= 1020;
			ELSE
				
				iState 							:= 30;
			END_IF
		END_IF
		
	30: 
		IF fbSQLResult.Release() THEN
			iState 								:= 999;	
		END_IF
		
	999:
		TON_Read.IN 	:= FALSE;
		Done			:= TRUE;
		Busy			:= FALSE;
		
 END_CASE 
 
IF iState > 1000 THEN
	Error 		:= TRUE;
	ErrorID	 	:= iState;
	Busy	 	:= FALSE;
	TON_Read.IN := FALSE;
	iState := -1;
END_IF

END_FUNCTION_BLOCK

// ---- FBs/Database/FB/FB_MSSQL_spGetPartHistoryByBatchName.TcPOU
FUNCTION_BLOCK FB_MSSQL_spGetPartHistoryByBatchName
VAR_INPUT
	Execute					: BOOL;
	Enable					: BOOL;
	Reset					: BOOL;
	sName					: STRING(50);
END_VAR
VAR_OUTPUT
	Error					: BOOL;
	ErrorID					: DINT;
	Done					: BOOL;
	Busy					: BOOL;
	tcMessage 				: I_TcMessage;
	Q_tElapsedTime			: TIME;
	Result					: STRING(DB.MAX_STRING_SIZE);
END_VAR
VAR
	RTRIG_Execute			: R_TRIG;
	RTRIG_Reset				: R_TRIG;
	iState					: INT := -1;
	TON_Read				: TON;
	Parameters				: STRING(50);
END_VAR
VAR_IN_OUT
	fbSQLResult				: FB_SQLResultEvt;
	fbSQLStoredProcedure	: FB_SQLStoredProcedureEvt;
END_VAR

RTRIG_Reset(CLK := Reset);
IF RTRIG_Reset.Q AND Execute AND Error AND NOT Busy THEN
	Execute := FALSE;
END_IF

RTRIG_Execute(CLK := Execute AND Enable);
IF(RTRIG_Execute.Q) THEN
	 Done							:= FALSE;
	 Error							:= FALSE;
	 ErrorID						:= 0;
	 
	 iState							:= 0;
ELSIF NOT Execute AND NOT Busy THEN
	Busy			:= FALSE;
	Done			:= FALSE;
	Error			:= FALSE;
	
	iState := -1;
END_IF
 
 // Elapsed Time
 TON_Read(PT:= T#5S);
 
 CASE iState OF
 
	 0:
	 		TON_Read.IN 						:= FALSE;
			Busy								:= TRUE;
			iState 								:= 10;
		
	10:
		IF fbSQLStoredProcedure.ExecuteDataReturn(pParameterStrc := ADR(Parameters), cbParameterStrc := SIZEOF(Parameters), pSQLDBResult := ADR(fbSqlResult)) THEN
			TON_Read.IN := TRUE;
			IF fbSQLStoredProcedure.bError THEN
				tcMessage := fbSQLStoredProcedure.ipTcResult;
				
				iState 							:= 1010;
			ELSE
				iState 							:= 20;
			END_IF    
		END_IF
		
	20:
		IF fbSQLResult.Read(0, fbSQLResult.nDataCount, ADR(Result), SIZEOF(Result), FALSE, TRUE) THEN
			IF fbSQLResult.bError THEN
				iState 							:= 1020;
			ELSE
				
				iState 							:= 30;
			END_IF
		END_IF
		
	30: 
		IF fbSQLResult.Release() THEN
			iState 								:= 999;	
		END_IF
		
	999:
		TON_Read.IN 	:= FALSE;
		Done			:= TRUE;
		Busy			:= FALSE;
		
 END_CASE 
 
IF iState > 1000 THEN
	Error 		:= TRUE;
	ErrorID	 	:= iState;
	Busy	 	:= FALSE;
	TON_Read.IN := FALSE;
	iState := -1;
END_IF

END_FUNCTION_BLOCK

// ---- FBs/Database/FB/FB_MSSQL_spGetSideCode.TcPOU
FUNCTION_BLOCK FB_MSSQL_spGetSideCode
VAR_INPUT
	Execute					: BOOL;
	Enable					: BOOL;
	Reset					: BOOL;
	CodeSchema				: STRING(50);
	SideBar					: STRING(50);
END_VAR
VAR_OUTPUT
	Error					: BOOL;
	ErrorID					: DINT;
	Done					: BOOL;
	Busy					: BOOL;
	tcMessage 				: I_TcMessage;
	Q_tElapsedTime			: TIME;
	Result					: STRING(DB.MAX_STRING_SIZE);
END_VAR
VAR
	RTRIG_Execute			: R_TRIG;
	RTRIG_Reset				: R_TRIG;
	iState					: INT := -1;
	TON_Read				: TON;
	Parameters					: DUT_GetBitting;
END_VAR
VAR_IN_OUT
	fbSQLResult				: FB_SQLResultEvt;
	fbSQLStoredProcedure	: FB_SQLStoredProcedureEvt;
END_VAR

RTRIG_Reset(CLK := Reset);
IF RTRIG_Reset.Q AND Execute AND Error AND NOT Busy THEN
	Execute := FALSE;
END_IF

RTRIG_Execute(CLK := Execute AND Enable);
IF(RTRIG_Execute.Q) THEN
	 Done							:= FALSE;
	 Error							:= FALSE;
	 ErrorID						:= 0;
	 
	 iState							:= 0;
ELSIF NOT Execute AND NOT Busy THEN
	Busy			:= FALSE;
	Done			:= FALSE;
	Error			:= FALSE;
	
	iState := -1;
END_IF
 
 // Elapsed Time
 TON_Read(PT:= T#5S);
 
 CASE iState OF
 
	 0:
	 		TON_Read.IN 						:= FALSE;
			Busy								:= TRUE;
			iState 								:= 10;
		
	10:
		IF fbSQLStoredProcedure.ExecuteDataReturn(pParameterStrc := ADR(Parameters), cbParameterStrc:= SIZEOF(Parameters), pSQLDBResult := ADR(fbSqlResult)) THEN
			TON_Read.IN := TRUE;
			IF fbSQLStoredProcedure.bError THEN
				tcMessage := fbSQLStoredProcedure.ipTcResult;
				
				iState 							:= 1010;
			ELSE
				iState 							:= 20;
			END_IF    
		END_IF
		
	20:
		IF fbSQLResult.Read(0, fbSQLResult.nDataCount, ADR(Result), SIZEOF(Result), FALSE, TRUE) THEN
			IF fbSQLResult.bError THEN
				iState 							:= 1020;
			ELSE
				
				iState 							:= 30;
			END_IF
		END_IF
		
	30: 
		IF fbSQLResult.Release() THEN
			iState 								:= 999;	
		END_IF
		
	999:
		TON_Read.IN 	:= FALSE;
		Done			:= TRUE;
		Busy			:= FALSE;
		
 END_CASE 
 
IF iState > 1000 THEN
	Error 		:= TRUE;
	ErrorID	 	:= iState;
	Busy	 	:= FALSE;
	TON_Read.IN := FALSE;
	iState := -1;
END_IF

END_FUNCTION_BLOCK

// ---- FBs/Database/FB/FB_MSSQL_spGetOrigins.TcPOU
FUNCTION_BLOCK FB_MSSQL_spGetOrigins
VAR_INPUT
	Execute					: BOOL;
	Enable					: BOOL;
	Reset					: BOOL;
END_VAR
VAR_OUTPUT
	Error					: BOOL;
	ErrorID					: DINT;
	Done					: BOOL;
	Busy					: BOOL;
	tcMessage 				: I_TcMessage;
	Q_tElapsedTime			: TIME;
	Result					: STRING(DB.MAX_STRING_SIZE);
END_VAR
VAR
	RTRIG_Execute			: R_TRIG;
	RTRIG_Reset				: R_TRIG;
	iState					: INT := -1;
	TON_Read				: TON;
END_VAR
VAR_IN_OUT
	fbSQLResult				: FB_SQLResultEvt;
	fbSQLStoredProcedure	: FB_SQLStoredProcedureEvt;
END_VAR

RTRIG_Reset(CLK := Reset);
IF RTRIG_Reset.Q AND Execute AND Error AND NOT Busy THEN
	Execute := FALSE;
END_IF

RTRIG_Execute(CLK := Execute AND Enable);
IF(RTRIG_Execute.Q) THEN
	 Done							:= FALSE;
	 Error							:= FALSE;
	 ErrorID						:= 0;
	 
	 iState							:= 0;
ELSIF NOT Execute AND NOT Busy THEN
	Busy			:= FALSE;
	Done			:= FALSE;
	Error			:= FALSE;
	
	iState := -1;
END_IF
 
 // Elapsed Time
 TON_Read(PT:= T#5S);
 
 CASE iState OF
 
	 0:
	 		TON_Read.IN 						:= FALSE;
			Busy								:= TRUE;
			iState 								:= 10;
		
	10:
		IF fbSQLStoredProcedure.ExecuteDataReturn(pParameterStrc := 0, cbParameterStrc:= 0, pSQLDBResult := ADR(fbSqlResult)) THEN
			TON_Read.IN := TRUE;
			IF fbSQLStoredProcedure.bError THEN
				tcMessage := fbSQLStoredProcedure.ipTcResult;
				
				iState 							:= 1010;
			ELSE
				iState 							:= 20;
			END_IF    
		END_IF
		
	20:
		IF fbSQLResult.Read(0, fbSQLResult.nDataCount, ADR(Result), SIZEOF(Result), FALSE, TRUE) THEN
			IF fbSQLResult.bError THEN
				iState 							:= 1020;
			ELSE
			
				iState 							:= 30;
			END_IF
		END_IF
		
	30: 
		IF fbSQLResult.Release() THEN
			iState 								:= 999;	
		END_IF
		
	999:
		TON_Read.IN 	:= FALSE;
		Done			:= TRUE;
		Busy			:= FALSE;
		
 END_CASE 
 
IF iState > 1000 THEN
	Error 		:= TRUE;
	ErrorID	 	:= iState;
	Busy	 	:= FALSE;
	TON_Read.IN := FALSE;
	iState := -1;
END_IF

END_FUNCTION_BLOCK

// ---- FBs/Database/FB/FB_MSSQL_spGetOriginsByName.TcPOU
FUNCTION_BLOCK FB_MSSQL_spGetOriginsByName
VAR_INPUT
	Execute					: BOOL;
	Enable					: BOOL;
	Reset					: BOOL;
	sName					: STRING(50);
END_VAR
VAR_OUTPUT
	Error					: BOOL;
	ErrorID					: DINT;
	Done					: BOOL;
	Busy					: BOOL;
	tcMessage 				: I_TcMessage;
	Q_tElapsedTime			: TIME;
	Result					: STRING(DB.MAX_STRING_SIZE);
END_VAR
VAR
	RTRIG_Execute			: R_TRIG;
	RTRIG_Reset				: R_TRIG;
	iState					: INT := -1;
	TON_Read				: TON;
	Parameters				: DUT_GetResourcesByName;
END_VAR
VAR_IN_OUT
	fbSQLResult				: FB_SQLResultEvt;
	fbSQLStoredProcedure	: FB_SQLStoredProcedureEvt;
END_VAR

RTRIG_Reset(CLK := Reset);
IF RTRIG_Reset.Q AND Execute AND Error AND NOT Busy THEN
	Execute := FALSE;
END_IF

Parameters.ResourceName :=  sName;
RTRIG_Execute(CLK := Execute AND Enable);
IF(RTRIG_Execute.Q) THEN
	 Done							:= FALSE;
	 Error							:= FALSE;
	 ErrorID						:= 0;
	 TON_Read.IN 						:= FALSE;
	 
	 iState							:= 0;
ELSIF NOT Execute AND NOT Busy THEN
	Busy			:= FALSE;
	Done			:= FALSE;
	Error			:= FALSE;
	
	iState := -1;
END_IF
 
 // Elapsed Time
 TON_Read(PT:= T#5S);
 
 CASE iState OF
 
	 0:
			Busy								:= TRUE;
			TON_Read.IN := TRUE;
			iState 								:= 10;
		
	10:
		IF fbSQLStoredProcedure.ExecuteDataReturn(pParameterStrc := ADR(Parameters), cbParameterStrc:= SIZEOF(Parameters), pSQLDBResult := ADR(fbSqlResult)) THEN
			
			IF fbSQLStoredProcedure.bError THEN
				tcMessage := fbSQLStoredProcedure.ipTcResult;
				
				iState 							:= 1010;
			ELSE
				iState 							:= 20;
			END_IF    
		END_IF
		
	20:
		IF fbSQLResult.Read(0, fbSQLResult.nDataCount, ADR(Result), SIZEOF(Result), FALSE, TRUE) THEN
			IF fbSQLResult.bError THEN
				iState 							:= 1020;
			ELSE
				
				iState 							:= 30;
			END_IF
		END_IF
		
	30: 
		IF fbSQLResult.Release() THEN
			Q_tElapsedTime := TON_Read.ET;
			iState 								:= 999;	
		END_IF
		
	999:
		TON_Read.IN 	:= FALSE;
		Done			:= TRUE;
		Busy			:= FALSE;
		
 END_CASE 
 
IF iState > 1000 THEN
	Error 		:= TRUE;
	ErrorID	 	:= iState;
	Busy	 	:= FALSE;
	TON_Read.IN := FALSE;
	iState := -1;
END_IF

END_FUNCTION_BLOCK

// ---- FBs/Database/FB/FB_MSSQL_spGetOriginsBySide.TcPOU
FUNCTION_BLOCK FB_MSSQL_spGetOriginsBySide
VAR_INPUT
	Execute					: BOOL;
	Enable					: BOOL;
	Reset					: BOOL;
	Side					: DINT;
END_VAR
VAR_OUTPUT
	Error					: BOOL;
	ErrorID					: DINT;
	Done					: BOOL;
	Busy					: BOOL;
	tcMessage 				: I_TcMessage;
	Q_tElapsedTime			: TIME;
	Result					: STRING(DB.MAX_STRING_SIZE);
END_VAR
VAR
	RTRIG_Execute			: R_TRIG;
	RTRIG_Reset				: R_TRIG;
	iState					: INT := -1;
	TON_Read				: TON;
END_VAR
VAR_IN_OUT
	fbSQLResult				: FB_SQLResultEvt;
	fbSQLStoredProcedure	: FB_SQLStoredProcedureEvt;
END_VAR

RTRIG_Reset(CLK := Reset);
IF RTRIG_Reset.Q AND Execute AND Error AND NOT Busy THEN
	Execute := FALSE;
END_IF

RTRIG_Execute(CLK := Execute AND Enable);
IF(RTRIG_Execute.Q) THEN
	 Done							:= FALSE;
	 Error							:= FALSE;
	 ErrorID						:= 0;
	 TON_Read.IN 						:= FALSE;
	 
	 iState							:= 0;
ELSIF NOT Execute AND NOT Busy THEN
	Busy			:= FALSE;
	Done			:= FALSE;
	Error			:= FALSE;
	
	iState := -1;
END_IF
 
 // Elapsed Time
 TON_Read(PT:= T#5S);
 
 CASE iState OF
 
	 0:
			Busy								:= TRUE;
			TON_Read.IN := TRUE;
			iState 								:= 10;
		
	10:
		IF fbSQLStoredProcedure.ExecuteDataReturn(pParameterStrc := ADR(Side), cbParameterStrc:= SIZEOF(Side), pSQLDBResult := ADR(fbSqlResult)) THEN
			
			IF fbSQLStoredProcedure.bError THEN
				tcMessage := fbSQLStoredProcedure.ipTcResult;
				
				iState 							:= 1010;
			ELSE
				iState 							:= 20;
			END_IF    
		END_IF
		
	20:
		IF fbSQLResult.Read(0, fbSQLResult.nDataCount, ADR(Result), SIZEOF(Result), FALSE, TRUE) THEN
			IF fbSQLResult.bError THEN
				iState 							:= 1020;
			ELSE
				
				iState 							:= 30;
			END_IF
		END_IF
		
	30: 
		IF fbSQLResult.Release() THEN
			Q_tElapsedTime := TON_Read.ET;
			iState 								:= 999;	
		END_IF
		
	999:
		TON_Read.IN 	:= FALSE;
		Done			:= TRUE;
		Busy			:= FALSE;
		
 END_CASE 
 
IF iState > 1000 THEN
	Error 		:= TRUE;
	ErrorID	 	:= iState;
	Busy	 	:= FALSE;
	TON_Read.IN := FALSE;
	iState := -1;
END_IF

END_FUNCTION_BLOCK

// ---- FBs/Database/FB/FB_MSSQL_spGetCutters.TcPOU
FUNCTION_BLOCK FB_MSSQL_spGetCutters
VAR_INPUT
	Execute					: BOOL;
	Enable					: BOOL;
	Reset					: BOOL;
END_VAR
VAR_OUTPUT
	Error					: BOOL;
	ErrorID					: DINT;
	Done					: BOOL;
	Busy					: BOOL;
	tcMessage 				: I_TcMessage;
	Q_tElapsedTime			: TIME;
	Result					: STRING(DB.MAX_STRING_SIZE);
END_VAR
VAR
	RTRIG_Execute			: R_TRIG;
	RTRIG_Reset				: R_TRIG;
	iState					: INT := -1;
	TON_Read				: TON;
END_VAR
VAR_IN_OUT
	fbSQLResult				: FB_SQLResultEvt;
	fbSQLStoredProcedure	: FB_SQLStoredProcedureEvt;
END_VAR

RTRIG_Reset(CLK := Reset);
IF RTRIG_Reset.Q AND Execute AND Error AND NOT Busy THEN
	Execute := FALSE;
END_IF

RTRIG_Execute(CLK := Execute AND Enable);
IF(RTRIG_Execute.Q) THEN
	 Done							:= FALSE;
	 Error							:= FALSE;
	 ErrorID						:= 0;
	 
	 iState							:= 0;
ELSIF NOT Execute AND NOT Busy THEN
	Busy			:= FALSE;
	Done			:= FALSE;
	Error			:= FALSE;
	
	iState := -1;
END_IF
 
 // Elapsed Time
 TON_Read(PT:= T#5S);
 
 CASE iState OF
 
	 0:
	 		TON_Read.IN 						:= FALSE;
			Busy								:= TRUE;
			iState 								:= 10;
		
	10:
		IF fbSQLStoredProcedure.ExecuteDataReturn(pParameterStrc := 0, cbParameterStrc:= 0, pSQLDBResult := ADR(fbSqlResult)) THEN
			TON_Read.IN := TRUE;
			IF fbSQLStoredProcedure.bError THEN
				tcMessage := fbSQLStoredProcedure.ipTcResult;
				
				iState 							:= 1010;
			ELSE
				iState 							:= 20;
			END_IF    
		END_IF
		
	20:
		IF fbSQLResult.Read(0, fbSQLResult.nDataCount, ADR(Result), SIZEOF(Result), FALSE, TRUE) THEN
			IF fbSQLResult.bError THEN
				iState 							:= 1020;
			ELSE
			
				iState 							:= 30;
			END_IF
		END_IF
		
	30: 
		IF fbSQLResult.Release() THEN
			iState 								:= 999;	
		END_IF
		
	999:
		TON_Read.IN 	:= FALSE;
		Done			:= TRUE;
		Busy			:= FALSE;
		
 END_CASE 
 
IF iState > 1000 THEN
	Error 		:= TRUE;
	ErrorID	 	:= iState;
	Busy	 	:= FALSE;
	TON_Read.IN := FALSE;
	iState := -1;
END_IF

END_FUNCTION_BLOCK

// ---- FBs/Database/FB/FB_MSSQL_spGetCuttersByName.TcPOU
FUNCTION_BLOCK FB_MSSQL_spGetCuttersByName
VAR_INPUT
	Execute					: BOOL;
	Enable					: BOOL;
	Reset					: BOOL;
	sName					: STRING(50);
END_VAR
VAR_OUTPUT
	Error					: BOOL;
	ErrorID					: DINT;
	Done					: BOOL;
	Busy					: BOOL;
	tcMessage 				: I_TcMessage;
	Q_tElapsedTime			: TIME;
	Result					: STRING(DB.MAX_STRING_SIZE);
END_VAR
VAR
	RTRIG_Execute			: R_TRIG;
	RTRIG_Reset				: R_TRIG;
	iState					: INT := -1;
	TON_Read				: TON;
	Parameters				: DUT_GetResourcesByName;
END_VAR
VAR_IN_OUT
	fbSQLResult				: FB_SQLResultEvt;
	fbSQLStoredProcedure	: FB_SQLStoredProcedureEvt;
END_VAR

RTRIG_Reset(CLK := Reset);
IF RTRIG_Reset.Q AND Execute AND Error AND NOT Busy THEN
	Execute := FALSE;
END_IF

Parameters.ResourceName :=  sName;
RTRIG_Execute(CLK := Execute AND Enable);
IF(RTRIG_Execute.Q) THEN
	 Done							:= FALSE;
	 Error							:= FALSE;
	 ErrorID						:= 0;
	 TON_Read.IN 						:= FALSE;
	 
	 iState							:= 0;
ELSIF NOT Execute AND NOT Busy THEN
	Busy			:= FALSE;
	Done			:= FALSE;
	Error			:= FALSE;
	
	iState := -1;
END_IF
 
 // Elapsed Time
 TON_Read(PT:= T#5S);
 
 CASE iState OF
 
	 0:
			Busy								:= TRUE;
			TON_Read.IN := TRUE;
			iState 								:= 10;
		
	10:
		IF fbSQLStoredProcedure.ExecuteDataReturn(pParameterStrc := ADR(Parameters), cbParameterStrc:= SIZEOF(Parameters), pSQLDBResult := ADR(fbSqlResult)) THEN
			
			IF fbSQLStoredProcedure.bError THEN
				tcMessage := fbSQLStoredProcedure.ipTcResult;
				
				iState 							:= 1010;
			ELSE
				iState 							:= 20;
			END_IF    
		END_IF
		
	20:
		IF fbSQLResult.Read(0, fbSQLResult.nDataCount, ADR(Result), SIZEOF(Result), FALSE, TRUE) THEN
			IF fbSQLResult.bError THEN
				iState 							:= 1020;
			ELSE
				
				iState 							:= 30;
			END_IF
		END_IF
		
	30: 
		IF fbSQLResult.Release() THEN
			Q_tElapsedTime := TON_Read.ET;
			iState 								:= 999;	
		END_IF
		
	999:
		TON_Read.IN 	:= FALSE;
		Done			:= TRUE;
		Busy			:= FALSE;
		
 END_CASE 
 
IF iState > 1000 THEN
	Error 		:= TRUE;
	ErrorID	 	:= iState;
	Busy	 	:= FALSE;
	TON_Read.IN := FALSE;
	iState := -1;
END_IF

END_FUNCTION_BLOCK

// ---- FBs/Database/FB/FB_MSSQL_spGetCuttersBySide.TcPOU
FUNCTION_BLOCK FB_MSSQL_spGetCuttersBySide
VAR_INPUT
	Execute					: BOOL;
	Enable					: BOOL;
	Reset					: BOOL;
	Side					: DINT;
END_VAR
VAR_OUTPUT
	Error					: BOOL;
	ErrorID					: DINT;
	Done					: BOOL;
	Busy					: BOOL;
	tcMessage 				: I_TcMessage;
	Q_tElapsedTime			: TIME;
	Result					: STRING(DB.MAX_STRING_SIZE);
END_VAR
VAR
	RTRIG_Execute			: R_TRIG;
	RTRIG_Reset				: R_TRIG;
	iState					: INT := -1;
	TON_Read				: TON;
END_VAR
VAR_IN_OUT
	fbSQLResult				: FB_SQLResultEvt;
	fbSQLStoredProcedure	: FB_SQLStoredProcedureEvt;
END_VAR

RTRIG_Reset(CLK := Reset);
IF RTRIG_Reset.Q AND Execute AND Error AND NOT Busy THEN
	Execute := FALSE;
END_IF

RTRIG_Execute(CLK := Execute AND Enable);
IF(RTRIG_Execute.Q) THEN
	 Done							:= FALSE;
	 Error							:= FALSE;
	 ErrorID						:= 0;
	 TON_Read.IN 						:= FALSE;
	 
	 iState							:= 0;
ELSIF NOT Execute AND NOT Busy THEN
	Busy			:= FALSE;
	Done			:= FALSE;
	Error			:= FALSE;
	
	iState := -1;
END_IF
 
 // Elapsed Time
 TON_Read(PT:= T#5S);
 
 CASE iState OF
 
	 0:
			Busy								:= TRUE;
			TON_Read.IN := TRUE;
			iState 								:= 10;
		
	10:
		IF fbSQLStoredProcedure.ExecuteDataReturn(pParameterStrc := ADR(Side), cbParameterStrc:= SIZEOF(Side), pSQLDBResult := ADR(fbSqlResult)) THEN
			
			IF fbSQLStoredProcedure.bError THEN
				tcMessage := fbSQLStoredProcedure.ipTcResult;
				
				iState 							:= 1010;
			ELSE
				iState 							:= 20;
			END_IF    
		END_IF
		
	20:
		IF fbSQLResult.Read(0, fbSQLResult.nDataCount, ADR(Result), SIZEOF(Result), FALSE, TRUE) THEN
			IF fbSQLResult.bError THEN
				iState 							:= 1020;
			ELSE
				
				iState 							:= 30;
			END_IF
		END_IF
		
	30: 
		IF fbSQLResult.Release() THEN
			Q_tElapsedTime := TON_Read.ET;
			iState 								:= 999;	
		END_IF
		
	999:
		TON_Read.IN 	:= FALSE;
		Done			:= TRUE;
		Busy			:= FALSE;
		
 END_CASE 
 
IF iState > 1000 THEN
	Error 		:= TRUE;
	ErrorID	 	:= iState;
	Busy	 	:= FALSE;
	TON_Read.IN := FALSE;
	iState := -1;
END_IF

END_FUNCTION_BLOCK

// ---- FBs/Database/FB/FB_MSSQL_spGetMillings.TcPOU
FUNCTION_BLOCK FB_MSSQL_spGetMillings
VAR_INPUT
	Execute					: BOOL;
	Enable					: BOOL;
	Reset					: BOOL;
END_VAR
VAR_OUTPUT
	Error					: BOOL;
	ErrorID					: DINT;
	Done					: BOOL;
	Busy					: BOOL;
	tcMessage 				: I_TcMessage;
	Q_tElapsedTime			: TIME;
	Result					: STRING(DB.MAX_STRING_SIZE);
END_VAR
VAR
	RTRIG_Execute			: R_TRIG;
	RTRIG_Reset				: R_TRIG;
	iState					: INT := -1;
	TON_Read				: TON;
END_VAR
VAR_IN_OUT
	fbSQLResult				: FB_SQLResultEvt;
	fbSQLStoredProcedure	: FB_SQLStoredProcedureEvt;
END_VAR

RTRIG_Reset(CLK := Reset);
IF RTRIG_Reset.Q AND Execute AND Error AND NOT Busy THEN
	Execute := FALSE;
END_IF

RTRIG_Execute(CLK := Execute AND Enable);
IF(RTRIG_Execute.Q) THEN
	 Done							:= FALSE;
	 Error							:= FALSE;
	 ErrorID						:= 0;
	 
	 iState							:= 0;
ELSIF NOT Execute AND NOT Busy THEN
	Busy			:= FALSE;
	Done			:= FALSE;
	Error			:= FALSE;
	
	iState := -1;
END_IF
 
 // Elapsed Time
 TON_Read(PT:= T#5S);
 
 CASE iState OF
 
	 0:
	 		TON_Read.IN 						:= FALSE;
			Busy								:= TRUE;
			iState 								:= 10;
		
	10:
		IF fbSQLStoredProcedure.ExecuteDataReturn(pParameterStrc := 0, cbParameterStrc:= 0, pSQLDBResult := ADR(fbSqlResult)) THEN
			TON_Read.IN := TRUE;
			IF fbSQLStoredProcedure.bError THEN
				tcMessage := fbSQLStoredProcedure.ipTcResult;
				
				iState 							:= 1010;
			ELSE
				iState 							:= 20;
			END_IF    
		END_IF
		
	20:
		IF fbSQLResult.Read(0, fbSQLResult.nDataCount, ADR(Result), SIZEOF(Result), FALSE, TRUE) THEN
			IF fbSQLResult.bError THEN
				iState 							:= 1020;
			ELSE
			
				iState 							:= 30;
			END_IF
		END_IF
		
	30: 
		IF fbSQLResult.Release() THEN
			iState 								:= 999;	
		END_IF
		
	999:
		TON_Read.IN 	:= FALSE;
		Done			:= TRUE;
		Busy			:= FALSE;
		
 END_CASE 
 
IF iState > 1000 THEN
	Error 		:= TRUE;
	ErrorID	 	:= iState;
	Busy	 	:= FALSE;
	TON_Read.IN := FALSE;
	iState := -1;
END_IF

END_FUNCTION_BLOCK

// ---- FBs/Database/FB/FB_MSSQL_spGetMillingsByName.TcPOU
FUNCTION_BLOCK FB_MSSQL_spGetMillingsByName
VAR_INPUT
	Execute					: BOOL;
	Enable					: BOOL;
	Reset					: BOOL;
	sName					: STRING(50);
END_VAR
VAR_OUTPUT
	Error					: BOOL;
	ErrorID					: DINT;
	Done					: BOOL;
	Busy					: BOOL;
	tcMessage 				: I_TcMessage;
	Q_tElapsedTime			: TIME;
	Result					: STRING(DB.MAX_STRING_SIZE);
END_VAR
VAR
	RTRIG_Execute			: R_TRIG;
	RTRIG_Reset				: R_TRIG;
	iState					: INT := -1;
	TON_Read				: TON;
	Parameters				: DUT_GetResourcesByName;
END_VAR
VAR_IN_OUT
	fbSQLResult				: FB_SQLResultEvt;
	fbSQLStoredProcedure	: FB_SQLStoredProcedureEvt;
END_VAR

RTRIG_Reset(CLK := Reset);
IF RTRIG_Reset.Q AND Execute AND Error AND NOT Busy THEN
	Execute := FALSE;
END_IF

Parameters.ResourceName :=  sName;
RTRIG_Execute(CLK := Execute AND Enable);
IF(RTRIG_Execute.Q) THEN
	 Done							:= FALSE;
	 Error							:= FALSE;
	 ErrorID						:= 0;
	 TON_Read.IN 						:= FALSE;
	 
	 iState							:= 0;
ELSIF NOT Execute AND NOT Busy THEN
	Busy			:= FALSE;
	Done			:= FALSE;
	Error			:= FALSE;
	
	iState := -1;
END_IF
 
 // Elapsed Time
 TON_Read(PT:= T#5S);
 
 CASE iState OF
 
	 0:
			Busy								:= TRUE;
			TON_Read.IN := TRUE;
			iState 								:= 10;
		
	10:
		IF fbSQLStoredProcedure.ExecuteDataReturn(pParameterStrc := ADR(Parameters), cbParameterStrc := SIZEOF(Parameters), pSQLDBResult := ADR(fbSqlResult)) THEN
			
			IF fbSQLStoredProcedure.bError THEN
				tcMessage := fbSQLStoredProcedure.ipTcResult;
				
				iState 							:= 1010;
			ELSE
				iState 							:= 20;
			END_IF    
		END_IF
		
	20:
		IF fbSQLResult.Read(0, fbSQLResult.nDataCount, ADR(Result), SIZEOF(Result), FALSE, TRUE) THEN
			IF fbSQLResult.bError THEN
				iState 							:= 1020;
			ELSE
				
				iState 							:= 30;
			END_IF
		END_IF
		
	30: 
		IF fbSQLResult.Release() THEN
			Q_tElapsedTime := TON_Read.ET;
			iState 								:= 999;	
		END_IF
		
	999:
		TON_Read.IN 	:= FALSE;
		Done			:= TRUE;
		Busy			:= FALSE;
		
 END_CASE 
 
IF iState > 1000 THEN
	Error 		:= TRUE;
	ErrorID	 	:= iState;
	Busy	 	:= FALSE;
	TON_Read.IN := FALSE;
	iState := -1;
END_IF

END_FUNCTION_BLOCK

// ---- FBs/Database/FB/FB_MSSQL_spGetMillingsByFamilyName.TcPOU
FUNCTION_BLOCK FB_MSSQL_spGetMillingsByFamilyName
VAR_INPUT
	Execute					: BOOL;
	Enable					: BOOL;
	Reset					: BOOL;
	sFamilyName				: STRING(50);
END_VAR
VAR_OUTPUT
	Error					: BOOL;
	ErrorID					: DINT;
	Done					: BOOL;
	Busy					: BOOL;
	tcMessage 				: I_TcMessage;
	Q_tElapsedTime			: TIME;
	Result					: STRING(DB.MAX_STRING_SIZE);
END_VAR
VAR
	RTRIG_Execute			: R_TRIG;
	RTRIG_Reset				: R_TRIG;
	iState					: INT := -1;
	TON_Read				: TON;
	Parameters				: DUT_GetResourcesByName;
END_VAR
VAR_IN_OUT
	fbSQLResult				: FB_SQLResultEvt;
	fbSQLStoredProcedure	: FB_SQLStoredProcedureEvt;
END_VAR

RTRIG_Reset(CLK := Reset);
IF RTRIG_Reset.Q AND Execute AND Error AND NOT Busy THEN
	Execute := FALSE;
END_IF

Parameters.ResourceName :=  sFamilyName;
RTRIG_Execute(CLK := Execute AND Enable);
IF(RTRIG_Execute.Q) THEN
	 Done							:= FALSE;
	 Error							:= FALSE;
	 ErrorID						:= 0;
	 TON_Read.IN 						:= FALSE;
	 
	 iState							:= 0;
ELSIF NOT Execute AND NOT Busy THEN
	Busy			:= FALSE;
	Done			:= FALSE;
	Error			:= FALSE;
	
	iState := -1;
END_IF
 
 // Elapsed Time
 TON_Read(PT:= T#5S);
 
 CASE iState OF
 
	 0:
			Busy								:= TRUE;
			TON_Read.IN := TRUE;
			iState 								:= 10;
		
	10:
		IF fbSQLStoredProcedure.ExecuteDataReturn(pParameterStrc := ADR(Parameters), cbParameterStrc:= SIZEOF(Parameters), pSQLDBResult := ADR(fbSqlResult)) THEN
			
			IF fbSQLStoredProcedure.bError THEN
				tcMessage := fbSQLStoredProcedure.ipTcResult;
				
				iState 							:= 1010;
			ELSE
				iState 							:= 20;
			END_IF    
		END_IF
		
	20:
		IF fbSQLResult.Read(0, fbSQLResult.nDataCount, ADR(Result), SIZEOF(Result), FALSE, TRUE) THEN
			IF fbSQLResult.bError THEN
				iState 							:= 1020;
			ELSE
				
				iState 							:= 30;
			END_IF
		END_IF
		
	30: 
		IF fbSQLResult.Release() THEN
			Q_tElapsedTime := TON_Read.ET;
			iState 								:= 999;	
		END_IF
		
	999:
		TON_Read.IN 	:= FALSE;
		Done			:= TRUE;
		Busy			:= FALSE;
		
 END_CASE 
 
IF iState > 1000 THEN
	Error 		:= TRUE;
	ErrorID	 	:= iState;
	Busy	 	:= FALSE;
	TON_Read.IN := FALSE;
	iState := -1;
END_IF

END_FUNCTION_BLOCK

// ---- FBs/Database/FB/FB_MSSQL_spGetResourcesByNameMilling.TcPOU
FUNCTION_BLOCK FB_MSSQL_spGetResourcesByNameMilling
VAR_INPUT
	Execute					: BOOL;
	Enable					: BOOL;
	Reset					: BOOL;
	sName					: STRING(50);
END_VAR
VAR_OUTPUT
	Error					: BOOL;
	ErrorID					: DINT;
	Done					: BOOL;
	Busy					: BOOL;
	tcMessage 				: I_TcMessage;
	Q_tElapsedTime			: TIME;
	Result					: STRING(DB.MAX_STRING_SIZE);
END_VAR
VAR
	RTRIG_Execute			: R_TRIG;
	RTRIG_Reset				: R_TRIG;
	iState					: INT := -1;
	TON_Read				: TON;
END_VAR
VAR_IN_OUT
	fbSQLResult				: FB_SQLResultEvt;
	fbSQLStoredProcedure	: FB_SQLStoredProcedureEvt;
END_VAR

RTRIG_Reset(CLK := Reset);
IF RTRIG_Reset.Q AND Execute AND Error AND NOT Busy THEN
	Execute := FALSE;
END_IF

RTRIG_Execute(CLK := Execute AND Enable);
IF(RTRIG_Execute.Q) THEN
	 Done							:= FALSE;
	 Error							:= FALSE;
	 ErrorID						:= 0;
	 TON_Read.IN 						:= FALSE;
	 
	 iState							:= 0;
ELSIF NOT Execute AND NOT Busy THEN
	Busy			:= FALSE;
	Done			:= FALSE;
	Error			:= FALSE;
	
	iState := -1;
END_IF
 
 // Elapsed Time
 TON_Read(PT:= T#5S);
 
 CASE iState OF
 
	 0:
			Busy								:= TRUE;
			TON_Read.IN := TRUE;
			iState 								:= 10;
		
	10:
		IF fbSQLStoredProcedure.ExecuteDataReturn(pParameterStrc := ADR(sName), cbParameterStrc:= SIZEOF(sName), pSQLDBResult := ADR(fbSqlResult)) THEN
			
			IF fbSQLStoredProcedure.bError THEN
				tcMessage := fbSQLStoredProcedure.ipTcResult;
				
				iState 							:= 1010;
			ELSE
				iState 							:= 20;
			END_IF    
		END_IF
		
	20:
		IF fbSQLResult.Read(0, fbSQLResult.nDataCount, ADR(Result), SIZEOF(Result), FALSE, TRUE) THEN
			IF fbSQLResult.bError THEN
				iState 							:= 1020;
			ELSE
				
				iState 							:= 30;
			END_IF
		END_IF
		
	30: 
		IF fbSQLResult.Release() THEN
			Q_tElapsedTime := TON_Read.ET;
			iState 								:= 999;	
		END_IF
		
	999:
		TON_Read.IN 	:= FALSE;
		Done			:= TRUE;
		Busy			:= FALSE;
		
 END_CASE 
 
IF iState > 1000 THEN
	Error 		:= TRUE;
	ErrorID	 	:= iState;
	Busy	 	:= FALSE;
	TON_Read.IN := FALSE;
	iState := -1;
END_IF

END_FUNCTION_BLOCK

// ---- FBs/Database/FB/FB_MSSQL_spGetOrderInfoList.TcPOU
FUNCTION_BLOCK FB_MSSQL_spGetOrderInfoList
VAR_INPUT
	Execute					: BOOL;
	Enable					: BOOL;
	Reset					: BOOL;
END_VAR
VAR_OUTPUT
	Error					: BOOL;
	ErrorID					: DINT;
	Done					: BOOL;
	Busy					: BOOL;
	tcMessage 				: I_TcMessage;
	Q_tElapsedTime			: TIME;
	Result					: STRING(DB.MAX_STRING_SIZE);
END_VAR
VAR
	RTRIG_Execute			: R_TRIG;
	RTRIG_Reset				: R_TRIG;
	iState					: INT := -1;
	TON_Read				: TON;
END_VAR
VAR_IN_OUT
	fbSQLResult				: FB_SQLResultEvt;
	fbSQLStoredProcedure	: FB_SQLStoredProcedureEvt;
END_VAR

RTRIG_Reset(CLK := Reset);
IF RTRIG_Reset.Q AND Execute AND Error AND NOT Busy THEN
	Execute := FALSE;
END_IF

RTRIG_Execute(CLK := Execute AND Enable);
IF(RTRIG_Execute.Q) THEN
	 Done							:= FALSE;
	 Error							:= FALSE;
	 ErrorID						:= 0;
	 
	 iState							:= 0;
ELSIF NOT Execute AND NOT Busy THEN
	Busy			:= FALSE;
	Done			:= FALSE;
	Error			:= FALSE;
	
	iState := -1;
END_IF
 
 // Elapsed Time
 TON_Read(PT:= T#5S);
 
 CASE iState OF
 
	 0:
	 		TON_Read.IN 						:= FALSE;
			Busy								:= TRUE;
			iState 								:= 10;
		
	10:
		IF fbSQLStoredProcedure.ExecuteDataReturn(pParameterStrc := 0, cbParameterStrc:= 0, pSQLDBResult := ADR(fbSqlResult)) THEN
			TON_Read.IN := TRUE;
			IF fbSQLStoredProcedure.bError THEN
				tcMessage := fbSQLStoredProcedure.ipTcResult;
				
				iState 							:= 1010;
			ELSE
				iState 							:= 20;
			END_IF    
		END_IF
		
	20:
		IF fbSQLResult.Read(0, fbSQLResult.nDataCount, ADR(Result), SIZEOF(Result), FALSE, TRUE) THEN
			IF fbSQLResult.bError THEN
				iState 							:= 1020;
			ELSE
				
				iState 							:= 30;
			END_IF
		END_IF
		
	30: 
		IF fbSQLResult.Release() THEN
			iState 								:= 999;	
		END_IF
		
